KUKA KRL program: EPS_2_251806_MH56A_A_20260212042253.src

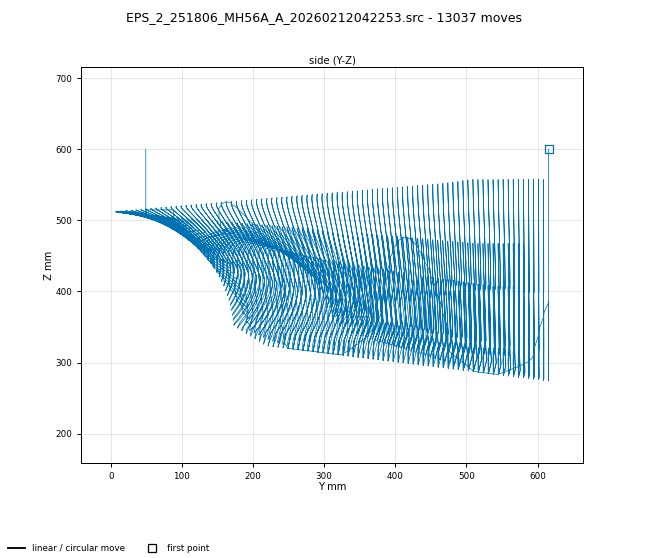
[picture p0: tool path of EPS_2_251806_MH56A_A_20260212042253.src, 13037 of 13039 moves have a stored position in this frame; points joined in program order, loops and branches not executed]
&ACCESS RVP
&REL 4
&COMMENT QRS 19112012
&PARAM EDITMASK = *
DEF PART()
EXT BAS (BAS_COMMAND :IN,REAL :IN )
INT I
BAS (#INITMOV,0 )

;KUKA QRS Post kuka4.cps  Date:22-06-2017 !

File_ID=3024

QRS_PRE_INIT()

;Init var - Until changes are made in qrs_pre_init
Outlet_Square_prg=0
Inlet_1_Square_prg=0
Inlet_2_Square_prg=0
Inlet_3_Square_prg=0
Inlet_4_Square_prg=0
Inlet_5_Square_prg=0

Outlet_1={X 0.000, Y 508.200, Z 408.000, B 0.000, E1 0.000 }
Inlet_1={X 0.000, Y 535.460, Z 257.000, B 0.000, E1 90.000 }
Inlet_2={X 0.000, Y 514.920, Z 318.000, B 0.000, E1 180.000 }
Outlet_1_type=299
Inlet_1_type=201
Inlet_2_type=299
;QRS#1=Sidecore dimensions
;QRS#2=300-12" PVC SDR 35
;QRS#3=200-8" PVC SDR 35
;QRS#4=300-12" PVC SDR 35
;QRS#5=
;QRS#6=
;QRS#7=
;QRS#8=
;QRS#9=16M PSX
;QRS#10=12-08 PSX
;QRS#11=16M PSX
;QRS#12=
;QRS#13=
;QRS#14=
;QRS#15=
;QRS#16=1220x127x838 2,75'
;QRS#17=EPS Height
;QRS#18=557,5
;QRS#19=*
;QRS#20= UPDATED VERSION 22-06-2017
;QRS#21=*
Outlet_Square=0150
Inlet_1_Square=0100
Inlet_2_Square=0150
Inlet_3_Square=0
Inlet_4_Square=0
Inlet_5_Square=0
Mill_Square=1
Outlet_Square_Prg=206
Inlet_1_Square_prg=204
Inlet_2_Square_prg=206

QRS_INIT()

$ADVANCE=5

; T1
PTP {E1 173.498,E2 173.498}
PTP {X 0,Y 615.498,A -85,B 0,C 180,E1 173.498,E2 173.498,E3 0,E4 0,E5 0,E6 0}
QRS_SPEED_INIT()
LIN {X 0,Y 615.498,Z 600,A -85,B 0,C 180,E1 173.498,E2 173.498,E3 0,E4 0,E5 0,E6 0} C_VEL
LIN {X 0,Y 615.498,Z 398.232,A -85,B 0,C 180,E1 173.498,E2 173.498} C_VEL
LIN {X 0,Y 615.498,Z 387.352,A -85,B 0,C 180,E1 173.498,E2 173.498} C_VEL
LIN {X 0,Y 615.496,Z 385.708,A -85,B 0,C 180,E1 173.418,E2 173.418} C_VEL
LIN {X 0,Y 615.498,Z 378.036,A -85,B 0,C 180,E1 172.455,E2 172.455} C_VEL
LIN {X 0,Y 615.498,Z 368.258,A -85,B 0,C 180,E1 171.463,E2 171.463} C_VEL
LIN {X 0,Y 615.498,Z 357.992,A -85,B 0,C 180,E1 170.636,E2 170.636} C_VEL
LIN {X 0,Y 615.489,Z 346.429,A -85,B 0,C 180,E1 169.889,E2 169.889} C_VEL
LIN {X 0,Y 615.479,Z 334.651,A -85,B 0,C 180,E1 169.296,E2 169.296} C_VEL
LIN {X 0,Y 615.485,Z 321.657,A -85,B 0,C 180,E1 168.807,E2 168.807} C_VEL
LIN {X 0,Y 615.492,Z 309.054,A -85,B 0,C 180,E1 168.473,E2 168.473} C_VEL
LIN {X 0,Y 615.49,Z 303.848,A -85,B 0,C 180,E1 168.369,E2 168.369} C_VEL
LIN {X 0,Y 615.48,Z 300.786,A -85,B 0,C 180,E1 166.071,E2 166.071} C_VEL
LIN {X 0,Y 615.479,Z 297.27,A -85,B 0,C 180,E1 163.413,E2 163.413} C_VEL
LIN {X 0,Y 615.488,Z 293.703,A -85,B 0,C 180,E1 160.662,E2 160.662} C_VEL
LIN {X 0,Y 615.494,Z 290.108,A -85,B 0,C 180,E1 157.864,E2 157.864} C_VEL
LIN {X 0,Y 615.499,Z 286.537,A -85,B 0,C 180,E1 155.009,E2 155.009} C_VEL
LIN {X 0,Y 615.485,Z 282.947,A -85,B 0,C 180,E1 152.085,E2 152.085} C_VEL
LIN {X 0,Y 615.497,Z 280.363,A -85,B 0,C 180,E1 149.84,E2 149.84} C_VEL
LIN {X 0,Y 615.449,Z 277.794,A -85,B 0,C 180,E1 147.54,E2 147.54} C_VEL
LIN {X 0,Y 615.456,Z 275.078,A -85,B 0,C 180,E1 145.183,E2 145.183} C_VEL
LIN {X 0,Y 615.496,Z 274.312,A -85,B 0,C 180,E1 144.166,E2 144.166} C_VEL
LIN {X 0,Y 615.481,Z 274.312,A -85,B 0,C 180,E1 141.931,E2 141.931} C_VEL
LIN {X 0,Y 615.483,Z 274.324,A -85,B 0,C 180,E1 139.393,E2 139.393} C_VEL
LIN {X 0,Y 615.467,Z 274.316,A -85,B 0,C 180,E1 136.753,E2 136.753} C_VEL
LIN {X 0,Y 615.492,Z 274.321,A -85,B 0,C 180,E1 133.998,E2 133.998} C_VEL
LIN {X 0,Y 615.443,Z 274.324,A -85,B 0,C 180,E1 131.478,E2 131.478} C_VEL
LIN {X 0,Y 615.464,Z 274.321,A -85,B 0,C 180,E1 130.609,E2 130.609} C_VEL
LIN {X 0,Y 615.478,Z 275.497,A -85,B 0,C 180,E1 129.751,E2 129.751} C_VEL
LIN {X 0,Y 615.477,Z 280.151,A -85,B 0,C 180,E1 126.935,E2 126.935} C_VEL
LIN {X 0,Y 615.455,Z 284.702,A -85,B 0,C 180,E1 124.024,E2 124.024} C_VEL
LIN {X 0,Y 615.486,Z 288.323,A -85,B 0,C 180,E1 121.686,E2 121.686} C_VEL
LIN {X 0,Y 615.494,Z 291.936,A -85,B 0,C 180,E1 119.406,E2 119.406} C_VEL
LIN {X 0,Y 615.488,Z 296.744,A -85,B 0,C 180,E1 116.444,E2 116.444} C_VEL
LIN {X 0,Y 615.478,Z 300.805,A -85,B 0,C 180,E1 114.006,E2 114.006} C_VEL
LIN {X 0,Y 615.491,Z 305.165,A -85,B 0,C 180,E1 111.432,E2 111.432} C_VEL
LIN {X 0,Y 615.488,Z 310.047,A -85,B 0,C 180,E1 108.604,E2 108.604} C_VEL
LIN {X 0,Y 615.489,Z 314.21,A -85,B 0,C 180,E1 106.3,E2 106.3} C_VEL
LIN {X 0,Y 615.499,Z 330.161,A -85,B 0,C 180,E1 106.036,E2 106.036} C_VEL
LIN {X 0,Y 615.493,Z 345.208,A -85,B 0,C 180,E1 105.65,E2 105.65} C_VEL
LIN {X 0,Y 615.479,Z 359.714,A -85,B 0,C 180,E1 105.142,E2 105.142} C_VEL
LIN {X 0,Y 615.489,Z 374.502,A -85,B 0,C 180,E1 104.473,E2 104.473} C_VEL
LIN {X 0,Y 615.496,Z 388.073,A -85,B 0,C 180,E1 103.706,E2 103.706} C_VEL
LIN {X 0,Y 615.496,Z 401.457,A -85,B 0,C 180,E1 102.782,E2 102.782} C_VEL
LIN {X 0,Y 615.495,Z 412.571,A -85,B 0,C 180,E1 101.861,E2 101.861} C_VEL
LIN {X 0,Y 615.493,Z 422.483,A -85,B 0,C 180,E1 100.89,E2 100.89} C_VEL
LIN {X 0,Y 615.495,Z 432.76,A -85,B 0,C 180,E1 99.696,E2 99.696} C_VEL
LIN {X 0,Y 615.49,Z 441.028,A -85,B 0,C 180,E1 98.537,E2 98.537} C_VEL
LIN {X 0,Y 615.491,Z 448.782,A -85,B 0,C 180,E1 97.216,E2 97.216} C_VEL
LIN {X 0,Y 615.499,Z 454.947,A -85,B 0,C 180,E1 95.899,E2 95.899} C_VEL
LIN {X 0,Y 615.489,Z 459.716,A -85,B 0,C 180,E1 94.585,E2 94.585} C_VEL
LIN {X 0,Y 615.491,Z 463.221,A -85,B 0,C 180,E1 93.273,E2 93.273} C_VEL
LIN {X 0,Y 615.5,Z 465.54,A -85,B 0,C 180,E1 91.963,E2 91.963} C_VEL
LIN {X 0,Y 615.491,Z 466.728,A -85,B 0,C 180,E1 90.654,E2 90.654} C_VEL
LIN {X 0,Y 615.492,Z 466.751,A -85,B 0,C 180,E1 89.346,E2 89.346} C_VEL
LIN {X 0,Y 615.5,Z 465.646,A -85,B 0,C 180,E1 88.037,E2 88.037} C_VEL
LIN {X 0,Y 615.494,Z 463.416,A -85,B 0,C 180,E1 86.727,E2 86.727} C_VEL
LIN {X 0,Y 615.49,Z 460.005,A -85,B 0,C 180,E1 85.416,E2 85.416} C_VEL
LIN {X 0,Y 615.499,Z 455.336,A -85,B 0,C 180,E1 84.102,E2 84.102} C_VEL
LIN {X 0,Y 615.49,Z 449.273,A -85,B 0,C 180,E1 82.785,E2 82.785} C_VEL
LIN {X 0,Y 615.493,Z 441.633,A -85,B 0,C 180,E1 81.464,E2 81.464} C_VEL
LIN {X 0,Y 615.496,Z 433.451,A -85,B 0,C 180,E1 80.304,E2 80.304} C_VEL
LIN {X 0,Y 615.495,Z 423.338,A -85,B 0,C 180,E1 79.109,E2 79.109} C_VEL
LIN {X 0,Y 615.497,Z 411.684,A -85,B 0,C 180,E1 77.972,E2 77.972} C_VEL
LIN {X 0,Y 615.498,Z 400.413,A -85,B 0,C 180,E1 77.051,E2 77.051} C_VEL
LIN {X 0,Y 615.498,Z 388.174,A -85,B 0,C 180,E1 76.21,E2 76.21} C_VEL
LIN {X 0,Y 615.495,Z 374.776,A -85,B 0,C 180,E1 75.451,E2 75.451} C_VEL
LIN {X 0,Y 615.478,Z 360.912,A -85,B 0,C 180,E1 74.816,E2 74.816} C_VEL
LIN {X 0,Y 615.496,Z 346.696,A -85,B 0,C 180,E1 74.308,E2 74.308} C_VEL
LIN {X 0,Y 615.496,Z 332.617,A -85,B 0,C 180,E1 73.931,E2 73.931} C_VEL
LIN {X 0,Y 615.494,Z 318.237,A -85,B 0,C 180,E1 73.667,E2 73.667} C_VEL
LIN {X 0,Y 615.493,Z 314.073,A -85,B 0,C 180,E1 73.601,E2 73.601} C_VEL
LIN {X 0,Y 615.489,Z 310.132,A -85,B 0,C 180,E1 71.354,E2 71.354} C_VEL
LIN {X 0,Y 615.485,Z 305.319,A -85,B 0,C 180,E1 68.568,E2 68.568} C_VEL
LIN {X 0,Y 615.48,Z 300.507,A -85,B 0,C 180,E1 65.728,E2 65.728} C_VEL
LIN {X 0,Y 615.498,Z 295.905,A -85,B 0,C 180,E1 62.953,E2 62.953} C_VEL
LIN {X 0,Y 615.477,Z 291.462,A -85,B 0,C 180,E1 60.207,E2 60.207} C_VEL
LIN {X 0,Y 615.492,Z 287.263,A -85,B 0,C 180,E1 57.543,E2 57.543} C_VEL
LIN {X 0,Y 615.477,Z 283.629,A -85,B 0,C 180,E1 55.184,E2 55.184} C_VEL
LIN {X 0,Y 615.485,Z 279.803,A -85,B 0,C 180,E1 52.758,E2 52.758} C_VEL
LIN {X 0,Y 615.484,Z 275.048,A -85,B 0,C 180,E1 49.912,E2 49.912} C_VEL
LIN {X 0,Y 615.465,Z 274.324,A -85,B 0,C 180,E1 49.392,E2 49.392} C_VEL
LIN {X 0,Y 615.463,Z 274.323,A -85,B 0,C 180,E1 46.753,E2 46.753} C_VEL
LIN {X 0,Y 615.485,Z 274.314,A -85,B 0,C 180,E1 43.997,E2 43.997} C_VEL
LIN {X 0,Y 615.467,Z 274.324,A -85,B 0,C 180,E1 41.092,E2 41.092} C_VEL
LIN {X 0,Y 615.434,Z 274.325,A -85,B 0,C 180,E1 38.908,E2 38.908} C_VEL
LIN {X 0,Y 615.483,Z 274.327,A -85,B 0,C 180,E1 36.425,E2 36.425} C_VEL
LIN {X 0,Y 615.49,Z 274.313,A -85,B 0,C 180,E1 34.022,E2 34.022} C_VEL
LIN {X 0,Y 615.47,Z 274.323,A -85,B 0,C 180,E1 31.083,E2 31.083} C_VEL
LIN {X 0,Y 615.454,Z 274.325,A -85,B 0,C 180,E1 28.445,E2 28.445} C_VEL
LIN {X 0,Y 615.461,Z 274.319,A -85,B 0,C 180,E1 25.564,E2 25.564} C_VEL
LIN {X 0,Y 615.483,Z 274.323,A -85,B 0,C 180,E1 22.845,E2 22.845} C_VEL
LIN {X 0,Y 615.496,Z 274.317,A -85,B 0,C 180,E1 20.033,E2 20.033} C_VEL
LIN {X 0,Y 615.436,Z 274.325,A -85,B 0,C 180,E1 17.272,E2 17.272} C_VEL
LIN {X 0,Y 615.493,Z 274.321,A -85,B 0,C 180,E1 14.549,E2 14.549} C_VEL
LIN {X 0,Y 615.479,Z 274.318,A -85,B 0,C 180,E1 11.861,E2 11.861} C_VEL
LIN {X 0,Y 615.458,Z 274.322,A -85,B 0,C 180,E1 9.199,E2 9.199} C_VEL
LIN {X 0,Y 615.479,Z 274.325,A -85,B 0,C 180,E1 6.557,E2 6.557} C_VEL
LIN {X 0,Y 615.461,Z 274.319,A -85,B 0,C 180,E1 3.929,E2 3.929} C_VEL
LIN {X 0,Y 615.492,Z 274.324,A -85,B 0,C 180,E1 1.309,E2 1.309} C_VEL
LIN {X 0,Y 615.484,Z 274.315,A -85,B 0,C 180,E1 -1.309,E2 -1.309} C_VEL
LIN {X 0,Y 615.458,Z 274.325,A -85,B 0,C 180,E1 -3.929,E2 -3.929} C_VEL
LIN {X 0,Y 615.462,Z 274.324,A -85,B 0,C 180,E1 -6.557,E2 -6.557} C_VEL
LIN {X 0,Y 615.492,Z 274.313,A -85,B 0,C 180,E1 -9.199,E2 -9.199} C_VEL
LIN {X 0,Y 615.489,Z 274.326,A -85,B 0,C 180,E1 -11.861,E2 -11.861} C_VEL
LIN {X 0,Y 615.437,Z 274.325,A -85,B 0,C 180,E1 -14.55,E2 -14.55} C_VEL
LIN {X 0,Y 615.491,Z 274.317,A -85,B 0,C 180,E1 -17.27,E2 -17.27} C_VEL
LIN {X 0,Y 615.484,Z 274.322,A -85,B 0,C 180,E1 -20.033,E2 -20.033} C_VEL
LIN {X 0,Y 615.477,Z 274.316,A -85,B 0,C 180,E1 -22.845,E2 -22.845} C_VEL
LIN {X 0,Y 615.446,Z 274.325,A -85,B 0,C 180,E1 -25.718,E2 -25.718} C_VEL
LIN {X 0,Y 615.448,Z 274.323,A -85,B 0,C 180,E1 -27.917,E2 -27.917} C_VEL
LIN {X 0,Y 615.492,Z 274.324,A -85,B 0,C 180,E1 -30.16,E2 -30.16} C_VEL
LIN {X 0,Y 615.473,Z 274.318,A -85,B 0,C 180,E1 -32.458,E2 -32.458} C_VEL
LIN {X 0,Y 615.487,Z 274.317,A -85,B 0,C 180,E1 -34.815,E2 -34.815} C_VEL
LIN {X 0,Y 615.457,Z 274.325,A -85,B 0,C 180,E1 -37.244,E2 -37.244} C_VEL
LIN {X 0,Y 615.485,Z 274.324,A -85,B 0,C 180,E1 -40.089,E2 -40.089} C_VEL
LIN {X 0,Y 615.488,Z 274.315,A -85,B 0,C 180,E1 -43.047,E2 -43.047} C_VEL
LIN {X 0,Y 615.449,Z 274.323,A -85,B 0,C 180,E1 -45.847,E2 -45.847} C_VEL
LIN {X 0,Y 615.496,Z 274.325,A -85,B 0,C 180,E1 -48.527,E2 -48.527} C_VEL
LIN {X 0,Y 615.468,Z 274.318,A -85,B 0,C 180,E1 -51.094,E2 -51.094} C_VEL
LIN {X 0,Y 615.483,Z 274.328,A -85,B 0,C 180,E1 -53.575,E2 -53.575} C_VEL
LIN {X 0,Y 615.468,Z 274.414,A -85,B 0,C 180,E1 -56.221,E2 -56.221} C_VEL
LIN {X 0,Y 615.492,Z 293.302,A -85,B 0,C 180,E1 -59.081,E2 -59.081} C_VEL
LIN {X 0,Y 615.485,Z 311.921,A -85,B 0,C 180,E1 -61.816,E2 -61.816} C_VEL
LIN {X 0,Y 615.492,Z 331.172,A -85,B 0,C 180,E1 -64.574,E2 -64.574} C_VEL
LIN {X 0,Y 615.499,Z 351.406,A -85,B 0,C 180,E1 -67.406,E2 -67.406} C_VEL
LIN {X 0,Y 615.485,Z 372.62,A -85,B 0,C 180,E1 -70.315,E2 -70.315} C_VEL
LIN {X 0,Y 615.491,Z 394.335,A -85,B 0,C 180,E1 -73.243,E2 -73.243} C_VEL
LIN {X 0,Y 615.484,Z 397.037,A -85,B 0,C 180,E1 -73.57,E2 -73.57} C_VEL
LIN {X 0,Y 615.478,Z 415.651,A -85,B 0,C 180,E1 -73.832,E2 -73.832} C_VEL
LIN {X 0,Y 615.491,Z 430.771,A -85,B 0,C 180,E1 -74.18,E2 -74.18} C_VEL
LIN {X 0,Y 615.493,Z 445.307,A -85,B 0,C 180,E1 -74.647,E2 -74.647} C_VEL
LIN {X 0,Y 615.497,Z 458.613,A -85,B 0,C 180,E1 -75.198,E2 -75.198} C_VEL
LIN {X 0,Y 615.498,Z 472.397,A -85,B 0,C 180,E1 -75.91,E2 -75.91} C_VEL
LIN {X 0,Y 615.498,Z 485.154,A -85,B 0,C 180,E1 -76.715,E2 -76.715} C_VEL
LIN {X 0,Y 615.496,Z 497.294,A -85,B 0,C 180,E1 -77.638,E2 -77.638} C_VEL
LIN {X 0,Y 615.497,Z 508.355,A -85,B 0,C 180,E1 -78.64,E2 -78.64} C_VEL
LIN {X 0,Y 615.496,Z 519.07,A -85,B 0,C 180,E1 -79.806,E2 -79.806} C_VEL
LIN {X 0,Y 615.495,Z 527.989,A -85,B 0,C 180,E1 -80.967,E2 -80.967} C_VEL
LIN {X 0,Y 615.492,Z 535.394,A -85,B 0,C 180,E1 -82.125,E2 -82.125} C_VEL
LIN {X 0,Y 615.491,Z 542.273,A -85,B 0,C 180,E1 -83.443,E2 -83.443} C_VEL
LIN {X 0,Y 615.491,Z 547.666,A -85,B 0,C 180,E1 -84.759,E2 -84.759} C_VEL
LIN {X 0,Y 615.491,Z 551.741,A -85,B 0,C 180,E1 -86.072,E2 -86.072} C_VEL
LIN {X 0,Y 615.496,Z 554.6,A -85,B 0,C 180,E1 -87.382,E2 -87.382} C_VEL
LIN {X 0,Y 615.493,Z 556.307,A -85,B 0,C 180,E1 -88.692,E2 -88.692} C_VEL
LIN {X 0,Y 615.491,Z 556.889,A -85,B 0,C 180,E1 -90,E2 -90} C_VEL
LIN {X 0,Y 615.493,Z 556.306,A -85,B 0,C 180,E1 -91.309,E2 -91.309} C_VEL
LIN {X 0,Y 615.496,Z 554.599,A -85,B 0,C 180,E1 -92.618,E2 -92.618} C_VEL
LIN {X 0,Y 615.491,Z 551.74,A -85,B 0,C 180,E1 -93.929,E2 -93.929} C_VEL
LIN {X 0,Y 615.491,Z 547.665,A -85,B 0,C 180,E1 -95.241,E2 -95.241} C_VEL
LIN {X 0,Y 615.491,Z 542.153,A -85,B 0,C 180,E1 -96.581,E2 -96.581} C_VEL
LIN {X 0,Y 615.492,Z 535.392,A -85,B 0,C 180,E1 -97.876,E2 -97.876} C_VEL
LIN {X 0,Y 615.495,Z 526.807,A -85,B 0,C 180,E1 -99.199,E2 -99.199} C_VEL
LIN {X 0,Y 615.494,Z 517.665,A -85,B 0,C 180,E1 -100.361,E2 -100.361} C_VEL
LIN {X 0,Y 615.497,Z 508.352,A -85,B 0,C 180,E1 -101.36,E2 -101.36} C_VEL
LIN {X 0,Y 615.496,Z 497.291,A -85,B 0,C 180,E1 -102.363,E2 -102.363} C_VEL
LIN {X 0,Y 615.498,Z 485.15,A -85,B 0,C 180,E1 -103.285,E2 -103.285} C_VEL
LIN {X 0,Y 615.498,Z 472.404,A -85,B 0,C 180,E1 -104.09,E2 -104.09} C_VEL
LIN {X 0,Y 615.497,Z 458.606,A -85,B 0,C 180,E1 -104.803,E2 -104.803} C_VEL
LIN {X 0,Y 615.495,Z 444.178,A -85,B 0,C 180,E1 -105.396,E2 -105.396} C_VEL
LIN {X 0,Y 615.488,Z 429.242,A -85,B 0,C 180,E1 -105.863,E2 -105.863} C_VEL
LIN {X 0,Y 615.478,Z 413.885,A -85,B 0,C 180,E1 -106.201,E2 -106.201} C_VEL
LIN {X 0,Y 615.485,Z 396.634,A -85,B 0,C 180,E1 -106.45,E2 -106.45} C_VEL
LIN {X 0,Y 615.484,Z 376.453,A -85,B 0,C 180,E1 -109.165,E2 -109.165} C_VEL
LIN {X 0,Y 615.481,Z 355.997,A -85,B 0,C 180,E1 -111.96,E2 -111.96} C_VEL
LIN {X 0,Y 615.498,Z 335.525,A -85,B 0,C 180,E1 -114.811,E2 -114.811} C_VEL
LIN {X 0,Y 615.497,Z 316.332,A -85,B 0,C 180,E1 -117.545,E2 -117.545} C_VEL
LIN {X 0,Y 615.489,Z 297.138,A -85,B 0,C 180,E1 -120.35,E2 -120.35} C_VEL
LIN {X 0,Y 615.485,Z 279.225,A -85,B 0,C 180,E1 -123.041,E2 -123.041} C_VEL
LIN {X 0,Y 615.477,Z 274.321,A -85,B 0,C 180,E1 -123.809,E2 -123.809} C_VEL
LIN {X 0,Y 615.458,Z 274.325,A -85,B 0,C 180,E1 -126.427,E2 -126.427} C_VEL
LIN {X 0,Y 615.486,Z 274.319,A -85,B 0,C 180,E1 -129.062,E2 -129.062} C_VEL
LIN {X 0,Y 615.465,Z 274.324,A -85,B 0,C 180,E1 -132.078,E2 -132.078} C_VEL
LIN {X 0,Y 615.476,Z 274.325,A -85,B 0,C 180,E1 -134.151,E2 -134.151} C_VEL
LIN {X 0,Y 615.492,Z 274.32,A -85,B 0,C 180,E1 -136.953,E2 -136.953} C_VEL
LIN {X 0,Y 615.458,Z 274.325,A -85,B 0,C 180,E1 -139.915,E2 -139.915} C_VEL
LIN {X 0,Y 615.483,Z 274.328,A -85,B 0,C 180,E1 -141.989,E2 -141.989} C_VEL
LIN {X 0,Y 615.469,Z 274.325,A -85,B 0,C 180,E1 -144.383,E2 -144.383} C_VEL
LIN {X 0,Y 615.49,Z 277.219,A -85,B 0,C 180,E1 -146.764,E2 -146.764} C_VEL
LIN {X 0,Y 615.489,Z 279.778,A -85,B 0,C 180,E1 -149.08,E2 -149.08} C_VEL
LIN {X 0,Y 615.494,Z 282.195,A -85,B 0,C 180,E1 -151.549,E2 -151.549} C_VEL
LIN {X 0,Y 615.478,Z 285.525,A -85,B 0,C 180,E1 -154.284,E2 -154.284} C_VEL
LIN {X 0,Y 615.473,Z 288.213,A -85,B 0,C 180,E1 -156.443,E2 -156.443} C_VEL
LIN {X 0,Y 615.479,Z 290.901,A -85,B 0,C 180,E1 -158.568,E2 -158.568} C_VEL
LIN {X 0,Y 615.483,Z 294.526,A -85,B 0,C 180,E1 -161.397,E2 -161.397} C_VEL
LIN {X 0,Y 615.477,Z 298.053,A -85,B 0,C 180,E1 -164.095,E2 -164.095} C_VEL
LIN {X 0,Y 615.494,Z 301.626,A -85,B 0,C 180,E1 -166.799,E2 -166.799} C_VEL
LIN {X 0,Y 615.488,Z 303.841,A -85,B 0,C 180,E1 -168.452,E2 -168.452} C_VEL
LIN {X 0,Y 615.49,Z 318.757,A -85,B 0,C 180,E1 -168.807,E2 -168.807} C_VEL
LIN {X 0,Y 615.478,Z 331.473,A -85,B 0,C 180,E1 -169.251,E2 -169.251} C_VEL
LIN {X 0,Y 615.488,Z 343.258,A -85,B 0,C 180,E1 -169.806,E2 -169.806} C_VEL
LIN {X 0,Y 615.498,Z 354.349,A -85,B 0,C 180,E1 -170.47,E2 -170.47} C_VEL
LIN {X 0,Y 615.498,Z 363.323,A -85,B 0,C 180,E1 -171.133,E2 -171.133} C_VEL
LIN {X 0,Y 615.498,Z 372.535,A -85,B 0,C 180,E1 -171.959,E2 -171.959} C_VEL
LIN {X 0,Y 615.499,Z 381.392,A -85,B 0,C 180,E1 -172.943,E2 -172.943} C_VEL
LIN {X 0,Y 615.497,Z 388.624,A -85,B 0,C 180,E1 -173.937,E2 -173.937} C_VEL
LIN {X 0,Y 615.497,Z 393.458,A -85,B 0,C 180,E1 -174.759,E2 -174.759} C_VEL
LIN {X 0,Y 615.497,Z 398.157,A -85,B 0,C 180,E1 -175.744,E2 -175.744} C_VEL
LIN {X 0,Y 615.495,Z 401.755,A -85,B 0,C 180,E1 -176.727,E2 -176.727} C_VEL
LIN {X 0,Y 615.496,Z 403.615,A -85,B 0,C 180,E1 -177.382,E2 -177.382} C_VEL
LIN {X 0,Y 615.497,Z 405.034,A -85,B 0,C 180,E1 -178.037,E2 -178.037} C_VEL
LIN {X 0,Y 615.497,Z 406.641,A -85,B 0,C 180,E1 -179.346,E2 -179.346} C_VEL
LIN {X 0,Y 615.494,Z 406.884,A -85,B 0,C 180,E1 -180,E2 -180} C_VEL
LIN {X 0,Y 615.495,Z 406.705,A -85,B 0,C 180,E1 -180.654,E2 -180.654} C_VEL
LIN {X 0,Y 615.496,Z 405.183,A -85,B 0,C 180,E1 -181.963,E2 -181.963} C_VEL
LIN {X 0,Y 615.498,Z 403.841,A -85,B 0,C 180,E1 -182.618,E2 -182.618} C_VEL
LIN {X 0,Y 615.497,Z 400.994,A -85,B 0,C 180,E1 -183.601,E2 -183.601} C_VEL
LIN {X 0,Y 615.498,Z 397.134,A -85,B 0,C 180,E1 -184.585,E2 -184.585} C_VEL
LIN {X 0,Y 615.498,Z 392.151,A -85,B 0,C 180,E1 -185.57,E2 -185.57} C_VEL
LIN {X 0,Y 615.496,Z 385.708,A -85,B 0,C 180,E1 -186.582,E2 -186.582} C_VEL
LIN {X 0,Y 614.829,Z 382.526,A -85,B 0,C 180,E1 -187.031,E2 -187.031} C_VEL
LIN {X 0,Y 611.989,Z 376.953,A -85,B 0,C 180,E1 -187.748,E2 -187.748} C_VEL
LIN {X 0,Y 609.138,Z 370.678,A -85,B 0,C 180,E1 -188.429,E2 -188.429} C_VEL
LIN {X 0,Y 608.477,Z 366.436,A -85,B 0,C 180,E1 -188.819,E2 -188.819} C_VEL
LIN {X 0,Y 608.493,Z 355.888,A -85,B 0,C 180,E1 -189.641,E2 -189.641} C_VEL
LIN {X 0,Y 608.49,Z 345.11,A -85,B 0,C 180,E1 -190.313,E2 -190.313} C_VEL
LIN {X 0,Y 608.505,Z 332.825,A -85,B 0,C 180,E1 -190.912,E2 -190.912} C_VEL
LIN {X 0,Y 608.525,Z 320.464,A -85,B 0,C 180,E1 -191.365,E2 -191.365} C_VEL
LIN {X 0,Y 608.55,Z 308.153,A -85,B 0,C 180,E1 -191.681,E2 -191.681} C_VEL
LIN {X 0,Y 608.436,Z 304.336,A -85,B 0,C 180,E1 -191.768,E2 -191.768} C_VEL
LIN {X 0,Y 608.43,Z 301.322,A -85,B 0,C 180,E1 -194.038,E2 -194.038} C_VEL
LIN {X 0,Y 608.414,Z 297.716,A -85,B 0,C 180,E1 -196.785,E2 -196.785} C_VEL
LIN {X 0,Y 608.415,Z 294.109,A -85,B 0,C 180,E1 -199.572,E2 -199.572} C_VEL
LIN {X 0,Y 608.432,Z 290.425,A -85,B 0,C 180,E1 -202.469,E2 -202.469} C_VEL
LIN {X 0,Y 608.43,Z 286.896,A -85,B 0,C 180,E1 -205.302,E2 -205.302} C_VEL
LIN {X 0,Y 608.434,Z 283.29,A -85,B 0,C 180,E1 -208.268,E2 -208.268} C_VEL
LIN {X 0,Y 608.418,Z 280.772,A -85,B 0,C 180,E1 -210.548,E2 -210.548} C_VEL
LIN {X 0,Y 608.446,Z 277.236,A -85,B 0,C 180,E1 -213.672,E2 -213.672} C_VEL
LIN {X 0,Y 608.409,Z 275.386,A -85,B 0,C 180,E1 -215.28,E2 -215.28} C_VEL
LIN {X 0,Y 608.471,Z 275.313,A -85,B 0,C 180,E1 -217.746,E2 -217.746} C_VEL
LIN {X 0,Y 608.449,Z 275.317,A -85,B 0,C 180,E1 -220.328,E2 -220.328} C_VEL
LIN {X 0,Y 608.437,Z 275.319,A -85,B 0,C 180,E1 -222.961,E2 -222.961} C_VEL
LIN {X 0,Y 608.461,Z 275.316,A -85,B 0,C 180,E1 -225.736,E2 -225.736} C_VEL
LIN {X 0,Y 608.474,Z 275.32,A -85,B 0,C 180,E1 -227.939,E2 -227.939} C_VEL
LIN {X 0,Y 608.424,Z 275.497,A -85,B 0,C 180,E1 -229.694,E2 -229.694} C_VEL
LIN {X 0,Y 608.448,Z 279.803,A -85,B 0,C 180,E1 -232.252,E2 -232.252} C_VEL
LIN {X 0,Y 608.398,Z 283.677,A -85,B 0,C 180,E1 -234.719,E2 -234.719} C_VEL
LIN {X 0,Y 608.437,Z 287.9,A -85,B 0,C 180,E1 -237.481,E2 -237.481} C_VEL
LIN {X 0,Y 608.427,Z 292.186,A -85,B 0,C 180,E1 -240.218,E2 -240.218} C_VEL
LIN {X 0,Y 608.435,Z 296.336,A -85,B 0,C 180,E1 -242.801,E2 -242.801} C_VEL
LIN {X 0,Y 608.424,Z 300.657,A -85,B 0,C 180,E1 -245.427,E2 -245.427} C_VEL
LIN {X 0,Y 608.435,Z 304.288,A -85,B 0,C 180,E1 -247.593,E2 -247.593} C_VEL
LIN {X 0,Y 608.426,Z 309.128,A -85,B 0,C 180,E1 -250.428,E2 -250.428} C_VEL
LIN {X 0,Y 608.418,Z 313.969,A -85,B 0,C 180,E1 -253.215,E2 -253.215} C_VEL
LIN {X 0,Y 608.427,Z 314.471,A -85,B 0,C 180,E1 -253.501,E2 -253.501} C_VEL
LIN {X 0,Y 608.679,Z 319.163,A -85,B 0,C 180,E1 -253.583,E2 -253.583} C_VEL
LIN {X 0,Y 608.672,Z 334.421,A -85,B 0,C 180,E1 -253.879,E2 -253.879} C_VEL
LIN {X 0,Y 608.624,Z 349.147,A -85,B 0,C 180,E1 -254.297,E2 -254.297} C_VEL
LIN {X 0,Y 608.603,Z 363.748,A -85,B 0,C 180,E1 -254.854,E2 -254.854} C_VEL
LIN {X 0,Y 608.574,Z 378.302,A -85,B 0,C 180,E1 -255.564,E2 -255.564} C_VEL
LIN {X 0,Y 608.554,Z 391.99,A -85,B 0,C 180,E1 -256.39,E2 -256.39} C_VEL
LIN {X 0,Y 608.528,Z 404.719,A -85,B 0,C 180,E1 -257.324,E2 -257.324} C_VEL
LIN {X 0,Y 608.497,Z 416.269,A -85,B 0,C 180,E1 -258.339,E2 -258.339} C_VEL
LIN {X 0,Y 608.475,Z 425.99,A -85,B 0,C 180,E1 -259.35,E2 -259.35} C_VEL
LIN {X 0,Y 608.477,Z 435.522,A -85,B 0,C 180,E1 -260.526,E2 -260.526} C_VEL
LIN {X 0,Y 608.457,Z 443.455,A -85,B 0,C 180,E1 -261.698,E2 -261.698} C_VEL
LIN {X 0,Y 608.44,Z 450.869,A -85,B 0,C 180,E1 -263.034,E2 -263.034} C_VEL
LIN {X 0,Y 608.45,Z 456.757,A -85,B 0,C 180,E1 -264.365,E2 -264.365} C_VEL
LIN {X 0,Y 608.425,Z 460.239,A -85,B 0,C 180,E1 -265.362,E2 -265.362} C_VEL
LIN {X 0,Y 608.42,Z 463.788,A -85,B 0,C 180,E1 -266.689,E2 -266.689} C_VEL
LIN {X 0,Y 608.444,Z 466.138,A -85,B 0,C 180,E1 -268.014,E2 -268.014} C_VEL
LIN {X 0,Y 608.434,Z 467.336,A -85,B 0,C 180,E1 -269.338,E2 -269.338} C_VEL
LIN {X 0,Y 608.435,Z 467.361,A -85,B 0,C 180,E1 -270.662,E2 -270.662} C_VEL
LIN {X 0,Y 608.444,Z 466.244,A -85,B 0,C 180,E1 -271.986,E2 -271.986} C_VEL
LIN {X 0,Y 608.423,Z 463.984,A -85,B 0,C 180,E1 -273.311,E2 -273.311} C_VEL
LIN {X 0,Y 608.425,Z 460.527,A -85,B 0,C 180,E1 -274.638,E2 -274.638} C_VEL
LIN {X 0,Y 608.437,Z 455.8,A -85,B 0,C 180,E1 -275.967,E2 -275.967} C_VEL
LIN {X 0,Y 608.456,Z 449.67,A -85,B 0,C 180,E1 -277.299,E2 -277.299} C_VEL
LIN {X 0,Y 608.468,Z 441.956,A -85,B 0,C 180,E1 -278.636,E2 -278.636} C_VEL
LIN {X 0,Y 608.472,Z 433.712,A -85,B 0,C 180,E1 -279.809,E2 -279.809} C_VEL
LIN {X 0,Y 608.476,Z 424.059,A -85,B 0,C 180,E1 -280.958,E2 -280.958} C_VEL
LIN {X 0,Y 608.509,Z 413.666,A -85,B 0,C 180,E1 -281.999,E2 -281.999} C_VEL
LIN {X 0,Y 608.533,Z 401.606,A -85,B 0,C 180,E1 -283.015,E2 -283.015} C_VEL
LIN {X 0,Y 608.564,Z 388.182,A -85,B 0,C 180,E1 -283.95,E2 -283.95} C_VEL
LIN {X 0,Y 608.602,Z 374.764,A -85,B 0,C 180,E1 -284.717,E2 -284.717} C_VEL
LIN {X 0,Y 608.595,Z 359.846,A -85,B 0,C 180,E1 -285.403,E2 -285.403} C_VEL
LIN {X 0,Y 608.644,Z 344.624,A -85,B 0,C 180,E1 -285.938,E2 -285.938} C_VEL
LIN {X 0,Y 608.671,Z 329.703,A -85,B 0,C 180,E1 -286.321,E2 -286.321} C_VEL
LIN {X 0,Y 608.582,Z 315.359,A -85,B 0,C 180,E1 -286.565,E2 -286.565} C_VEL
LIN {X 0,Y 608.453,Z 314.481,A -85,B 0,C 180,E1 -286.582,E2 -286.582} C_VEL
LIN {X 0,Y 608.434,Z 310.495,A -85,B 0,C 180,E1 -288.87,E2 -288.87} C_VEL
LIN {X 0,Y 608.414,Z 305.651,A -85,B 0,C 180,E1 -291.693,E2 -291.693} C_VEL
LIN {X 0,Y 608.422,Z 301.527,A -85,B 0,C 180,E1 -294.141,E2 -294.141} C_VEL
LIN {X 0,Y 608.432,Z 297.174,A -85,B 0,C 180,E1 -296.775,E2 -296.775} C_VEL
LIN {X 0,Y 608.445,Z 293.541,A -85,B 0,C 180,E1 -299.021,E2 -299.021} C_VEL
LIN {X 0,Y 608.447,Z 289.908,A -85,B 0,C 180,E1 -301.318,E2 -301.318} C_VEL
LIN {X 0,Y 608.449,Z 286.214,A -85,B 0,C 180,E1 -303.731,E2 -303.731} C_VEL
LIN {X 0,Y 608.446,Z 282.555,A -85,B 0,C 180,E1 -306.092,E2 -306.092} C_VEL
LIN {X 0,Y 608.431,Z 278.602,A -85,B 0,C 180,E1 -308.591,E2 -308.591} C_VEL
LIN {X 0,Y 608.433,Z 275.622,A -85,B 0,C 180,E1 -310.327,E2 -310.327} C_VEL
LIN {X 0,Y 608.465,Z 275.316,A -85,B 0,C 180,E1 -312.335,E2 -312.335} C_VEL
LIN {X 0,Y 608.449,Z 275.317,A -85,B 0,C 180,E1 -314.796,E2 -314.796} C_VEL
LIN {X 0,Y 608.451,Z 275.322,A -85,B 0,C 180,E1 -317.04,E2 -317.04} C_VEL
LIN {X 0,Y 608.423,Z 275.32,A -85,B 0,C 180,E1 -319.694,E2 -319.694} C_VEL
LIN {X 0,Y 608.457,Z 275.318,A -85,B 0,C 180,E1 -322.253,E2 -322.253} C_VEL
LIN {X 0,Y 608.439,Z 275.318,A -85,B 0,C 180,E1 -324.722,E2 -324.722} C_VEL
LIN {X 0,Y 608.451,Z 275.321,A -85,B 0,C 180,E1 -327.12,E2 -327.12} C_VEL
LIN {X 0,Y 608.472,Z 275.317,A -85,B 0,C 180,E1 -330.028,E2 -330.028} C_VEL
LIN {X 0,Y 608.419,Z 275.32,A -85,B 0,C 180,E1 -332.804,E2 -332.804} C_VEL
LIN {X 0,Y 608.452,Z 275.321,A -85,B 0,C 180,E1 -335.429,E2 -335.429} C_VEL
LIN {X 0,Y 608.477,Z 275.316,A -85,B 0,C 180,E1 -338.309,E2 -338.309} C_VEL
LIN {X 0,Y 608.438,Z 275.317,A -85,B 0,C 180,E1 -341.13,E2 -341.13} C_VEL
LIN {X 0,Y 608.446,Z 275.319,A -85,B 0,C 180,E1 -343.906,E2 -343.906} C_VEL
LIN {X 0,Y 608.459,Z 275.318,A -85,B 0,C 180,E1 -346.643,E2 -346.643} C_VEL
LIN {X 0,Y 608.459,Z 275.315,A -85,B 0,C 180,E1 -349.35,E2 -349.35} C_VEL
LIN {X 0,Y 608.468,Z 275.32,A -85,B 0,C 180,E1 -352.033,E2 -352.033} C_VEL
LIN {X 0,Y 608.428,Z 275.319,A -85,B 0,C 180,E1 -354.698,E2 -354.698} C_VEL
LIN {X 0,Y 608.483,Z 275.314,A -85,B 0,C 180,E1 -357.352,E2 -357.352} C_VEL
LIN {X 0,Y 608.479,Z 275.316,A -85,B 0,C 180,E1 -360,E2 -360} C_VEL
LIN {X 0,Y 608.441,Z 275.317,A -85,B 0,C 180,E1 -362.648,E2 -362.648} C_VEL
LIN {X 0,Y 608.469,Z 275.32,A -85,B 0,C 180,E1 -365.302,E2 -365.302} C_VEL
LIN {X 0,Y 608.436,Z 275.318,A -85,B 0,C 180,E1 -367.967,E2 -367.967} C_VEL
LIN {X 0,Y 608.457,Z 275.317,A -85,B 0,C 180,E1 -370.65,E2 -370.65} C_VEL
LIN {X 0,Y 608.462,Z 275.319,A -85,B 0,C 180,E1 -373.356,E2 -373.356} C_VEL
LIN {X 0,Y 608.419,Z 275.319,A -85,B 0,C 180,E1 -376.095,E2 -376.095} C_VEL
LIN {X 0,Y 608.46,Z 275.318,A -85,B 0,C 180,E1 -378.869,E2 -378.869} C_VEL
LIN {X 0,Y 608.466,Z 275.318,A -85,B 0,C 180,E1 -381.692,E2 -381.692} C_VEL
LIN {X 0,Y 608.436,Z 275.318,A -85,B 0,C 180,E1 -384.572,E2 -384.572} C_VEL
LIN {X 0,Y 608.434,Z 275.318,A -85,B 0,C 180,E1 -387.519,E2 -387.519} C_VEL
LIN {X 0,Y 608.459,Z 275.318,A -85,B 0,C 180,E1 -389.97,E2 -389.97} C_VEL
LIN {X 0,Y 608.456,Z 275.315,A -85,B 0,C 180,E1 -392.88,E2 -392.88} C_VEL
LIN {X 0,Y 608.426,Z 275.326,A -85,B 0,C 180,E1 -395.279,E2 -395.279} C_VEL
LIN {X 0,Y 608.413,Z 275.32,A -85,B 0,C 180,E1 -397.75,E2 -397.75} C_VEL
LIN {X 0,Y 608.452,Z 275.322,A -85,B 0,C 180,E1 -400.329,E2 -400.329} C_VEL
LIN {X 0,Y 608.453,Z 275.316,A -85,B 0,C 180,E1 -402.96,E2 -402.96} C_VEL
LIN {X 0,Y 608.426,Z 275.32,A -85,B 0,C 180,E1 -405.739,E2 -405.739} C_VEL
LIN {X 0,Y 608.421,Z 275.32,A -85,B 0,C 180,E1 -407.935,E2 -407.935} C_VEL
LIN {X 0,Y 608.444,Z 275.318,A -85,B 0,C 180,E1 -410.706,E2 -410.706} C_VEL
LIN {X 0,Y 608.449,Z 275.318,A -85,B 0,C 180,E1 -413.085,E2 -413.085} C_VEL
LIN {X 0,Y 608.448,Z 275.359,A -85,B 0,C 180,E1 -415.918,E2 -415.918} C_VEL
LIN {X 0,Y 608.788,Z 279.231,A -85,B 0,C 180,E1 -416.548,E2 -416.548} C_VEL
LIN {X 0,Y 608.725,Z 297.141,A -85,B 0,C 180,E1 -419.277,E2 -419.277} C_VEL
LIN {X 0,Y 608.669,Z 315.054,A -85,B 0,C 180,E1 -421.932,E2 -421.932} C_VEL
LIN {X 0,Y 608.638,Z 334.247,A -85,B 0,C 180,E1 -424.707,E2 -424.707} C_VEL
LIN {X 0,Y 608.588,Z 353.971,A -85,B 0,C 180,E1 -427.494,E2 -427.494} C_VEL
LIN {X 0,Y 608.541,Z 373.913,A -85,B 0,C 180,E1 -430.257,E2 -430.257} C_VEL
LIN {X 0,Y 608.526,Z 395.665,A -85,B 0,C 180,E1 -433.218,E2 -433.218} C_VEL
LIN {X 0,Y 608.52,Z 396.72,A -85,B 0,C 180,E1 -433.36,E2 -433.36} C_VEL
LIN {X 0,Y 608.669,Z 405.711,A -85,B 0,C 180,E1 -433.488,E2 -433.488} C_VEL
LIN {X 0,Y 608.666,Z 420.715,A -85,B 0,C 180,E1 -433.746,E2 -433.746} C_VEL
LIN {X 0,Y 608.644,Z 435.302,A -85,B 0,C 180,E1 -434.126,E2 -434.126} C_VEL
LIN {X 0,Y 608.613,Z 449.794,A -85,B 0,C 180,E1 -434.641,E2 -434.641} C_VEL
LIN {X 0,Y 608.602,Z 463.861,A -85,B 0,C 180,E1 -435.283,E2 -435.283} C_VEL
LIN {X 0,Y 608.562,Z 477.448,A -85,B 0,C 180,E1 -436.05,E2 -436.05} C_VEL
LIN {X 0,Y 608.547,Z 489.855,A -85,B 0,C 180,E1 -436.9,E2 -436.9} C_VEL
LIN {X 0,Y 608.522,Z 501.275,A -85,B 0,C 180,E1 -437.832,E2 -437.832} C_VEL
LIN {X 0,Y 608.491,Z 512.651,A -85,B 0,C 180,E1 -438.937,E2 -438.937} C_VEL
LIN {X 0,Y 608.471,Z 523.371,A -85,B 0,C 180,E1 -440.191,E2 -440.191} C_VEL
LIN {X 0,Y 608.468,Z 531.655,A -85,B 0,C 180,E1 -441.364,E2 -441.364} C_VEL
LIN {X 0,Y 608.457,Z 539.427,A -85,B 0,C 180,E1 -442.701,E2 -442.701} C_VEL
LIN {X 0,Y 608.437,Z 545.608,A -85,B 0,C 180,E1 -444.033,E2 -444.033} C_VEL
LIN {X 0,Y 608.427,Z 550.383,A -85,B 0,C 180,E1 -445.362,E2 -445.362} C_VEL
LIN {X 0,Y 608.421,Z 553.886,A -85,B 0,C 180,E1 -446.689,E2 -446.689} C_VEL
LIN {X 0,Y 608.444,Z 556.191,A -85,B 0,C 180,E1 -448.014,E2 -448.014} C_VEL
LIN {X 0,Y 608.436,Z 557.351,A -85,B 0,C 180,E1 -449.338,E2 -449.338} C_VEL
LIN {X 0,Y 608.436,Z 557.351,A -85,B 0,C 180,E1 -450.662,E2 -450.662} C_VEL
LIN {X 0,Y 608.444,Z 556.191,A -85,B 0,C 180,E1 -451.986,E2 -451.986} C_VEL
LIN {X 0,Y 608.421,Z 553.885,A -85,B 0,C 180,E1 -453.311,E2 -453.311} C_VEL
LIN {X 0,Y 608.427,Z 550.382,A -85,B 0,C 180,E1 -454.638,E2 -454.638} C_VEL
LIN {X 0,Y 608.437,Z 545.607,A -85,B 0,C 180,E1 -455.967,E2 -455.967} C_VEL
LIN {X 0,Y 608.457,Z 539.425,A -85,B 0,C 180,E1 -457.3,E2 -457.3} C_VEL
LIN {X 0,Y 608.468,Z 531.653,A -85,B 0,C 180,E1 -458.636,E2 -458.636} C_VEL
LIN {X 0,Y 608.471,Z 523.369,A -85,B 0,C 180,E1 -459.809,E2 -459.809} C_VEL
LIN {X 0,Y 608.493,Z 512.647,A -85,B 0,C 180,E1 -461.064,E2 -461.064} C_VEL
LIN {X 0,Y 608.522,Z 501.272,A -85,B 0,C 180,E1 -462.168,E2 -462.168} C_VEL
LIN {X 0,Y 608.547,Z 489.851,A -85,B 0,C 180,E1 -463.1,E2 -463.1} C_VEL
LIN {X 0,Y 608.563,Z 477.443,A -85,B 0,C 180,E1 -463.95,E2 -463.95} C_VEL
LIN {X 0,Y 608.602,Z 463.854,A -85,B 0,C 180,E1 -464.718,E2 -464.718} C_VEL
LIN {X 0,Y 608.613,Z 449.786,A -85,B 0,C 180,E1 -465.36,E2 -465.36} C_VEL
LIN {X 0,Y 608.67,Z 434.558,A -85,B 0,C 180,E1 -465.895,E2 -465.895} C_VEL
LIN {X 0,Y 608.662,Z 419.159,A -85,B 0,C 180,E1 -466.288,E2 -466.288} C_VEL
LIN {X 0,Y 608.69,Z 403.969,A -85,B 0,C 180,E1 -466.535,E2 -466.535} C_VEL
LIN {X 0,Y 608.531,Z 396.984,A -85,B 0,C 180,E1 -466.624,E2 -466.624} C_VEL
LIN {X 0,Y 608.546,Z 376.47,A -85,B 0,C 180,E1 -469.392,E2 -469.392} C_VEL
LIN {X 0,Y 608.569,Z 357.277,A -85,B 0,C 180,E1 -472.044,E2 -472.044} C_VEL
LIN {X 0,Y 608.645,Z 336.804,A -85,B 0,C 180,E1 -474.927,E2 -474.927} C_VEL
LIN {X 0,Y 608.675,Z 317.611,A -85,B 0,C 180,E1 -477.694,E2 -477.694} C_VEL
LIN {X 0,Y 608.716,Z 298.418,A -85,B 0,C 180,E1 -480.531,E2 -480.531} C_VEL
LIN {X 0,Y 608.759,Z 281.784,A -85,B 0,C 180,E1 -483.059,E2 -483.059} C_VEL
LIN {X 0,Y 608.886,Z 277.387,A -85,B 0,C 180,E1 -483.793,E2 -483.793} C_VEL
LIN {X 0,Y 608.443,Z 275.323,A -85,B 0,C 180,E1 -484.221,E2 -484.221} C_VEL
LIN {X 0,Y 608.48,Z 275.32,A -85,B 0,C 180,E1 -487.16,E2 -487.16} C_VEL
LIN {X 0,Y 608.478,Z 275.316,A -85,B 0,C 180,E1 -489.439,E2 -489.439} C_VEL
LIN {X 0,Y 608.449,Z 275.321,A -85,B 0,C 180,E1 -492.333,E2 -492.333} C_VEL
LIN {X 0,Y 608.441,Z 275.32,A -85,B 0,C 180,E1 -494.798,E2 -494.798} C_VEL
LIN {X 0,Y 608.458,Z 275.319,A -85,B 0,C 180,E1 -497.666,E2 -497.666} C_VEL
LIN {X 0,Y 608.446,Z 275.324,A -85,B 0,C 180,E1 -500.706,E2 -500.706} C_VEL
LIN {X 0,Y 608.457,Z 275.32,A -85,B 0,C 180,E1 -503.085,E2 -503.085} C_VEL
LIN {X 0,Y 608.435,Z 275.52,A -85,B 0,C 180,E1 -504.722,E2 -504.722} C_VEL
LIN {X 0,Y 608.457,Z 278.611,A -85,B 0,C 180,E1 -507.121,E2 -507.121} C_VEL
LIN {X 0,Y 608.457,Z 281.698,A -85,B 0,C 180,E1 -510.031,E2 -510.031} C_VEL
LIN {X 0,Y 608.427,Z 284.083,A -85,B 0,C 180,E1 -512.481,E2 -512.481} C_VEL
LIN {X 0,Y 608.43,Z 287.687,A -85,B 0,C 180,E1 -515.428,E2 -515.428} C_VEL
LIN {X 0,Y 608.412,Z 291.291,A -85,B 0,C 180,E1 -518.306,E2 -518.306} C_VEL
LIN {X 0,Y 608.415,Z 293.994,A -85,B 0,C 180,E1 -520.428,E2 -520.428} C_VEL
LIN {X 0,Y 608.416,Z 297.599,A -85,B 0,C 180,E1 -523.215,E2 -523.215} C_VEL
LIN {X 0,Y 608.422,Z 301.257,A -85,B 0,C 180,E1 -526.002,E2 -526.002} C_VEL
LIN {X 0,Y 608.426,Z 304.443,A -85,B 0,C 180,E1 -528.338,E2 -528.338} C_VEL
LIN {X 0,Y 608.541,Z 318.137,A -85,B 0,C 180,E1 -528.656,E2 -528.656} C_VEL
LIN {X 0,Y 608.514,Z 330.053,A -85,B 0,C 180,E1 -529.062,E2 -529.062} C_VEL
LIN {X 0,Y 608.498,Z 341.869,A -85,B 0,C 180,E1 -529.603,E2 -529.603} C_VEL
LIN {X 0,Y 608.501,Z 353.291,A -85,B 0,C 180,E1 -530.275,E2 -530.275} C_VEL
LIN {X 0,Y 608.474,Z 363.585,A -85,B 0,C 180,E1 -531.029,E2 -531.029} C_VEL
LIN {X 0,Y 608.464,Z 372.85,A -85,B 0,C 180,E1 -531.866,E2 -531.866} C_VEL
LIN {X 0,Y 608.466,Z 381.824,A -85,B 0,C 180,E1 -532.867,E2 -532.867} C_VEL
LIN {X 0,Y 608.444,Z 389.056,A -85,B 0,C 180,E1 -533.867,E2 -533.867} C_VEL
LIN {X 0,Y 608.462,Z 393.935,A -85,B 0,C 180,E1 -534.698,E2 -534.698} C_VEL
LIN {X 0,Y 608.441,Z 398.678,A -85,B 0,C 180,E1 -535.694,E2 -535.694} C_VEL
LIN {X 0,Y 608.425,Z 402.312,A -85,B 0,C 180,E1 -536.689,E2 -536.689} C_VEL
LIN {X 0,Y 608.425,Z 404.191,A -85,B 0,C 180,E1 -537.352,E2 -537.352} C_VEL
LIN {X 0,Y 608.442,Z 405.627,A -85,B 0,C 180,E1 -538.014,E2 -538.014} C_VEL
LIN {X 0,Y 608.44,Z 407.252,A -85,B 0,C 180,E1 -539.338,E2 -539.338} C_VEL
LIN {X 0,Y 608.434,Z 407.495,A -85,B 0,C 180,E1 -540,E2 -540} C_VEL
LIN {X 0,Y 608.438,Z 407.315,A -85,B 0,C 180,E1 -540.662,E2 -540.662} C_VEL
LIN {X 0,Y 608.441,Z 405.776,A -85,B 0,C 180,E1 -541.986,E2 -541.986} C_VEL
LIN {X 0,Y 608.426,Z 404.418,A -85,B 0,C 180,E1 -542.648,E2 -542.648} C_VEL
LIN {X 0,Y 608.45,Z 401.541,A -85,B 0,C 180,E1 -543.642,E2 -543.642} C_VEL
LIN {X 0,Y 608.433,Z 397.642,A -85,B 0,C 180,E1 -544.638,E2 -544.638} C_VEL
LIN {X 0,Y 608.45,Z 392.612,A -85,B 0,C 180,E1 -545.634,E2 -545.634} C_VEL
LIN {X 0,Y 608.441,Z 386.294,A -85,B 0,C 180,E1 -546.633,E2 -546.633} C_VEL
LIN {X 0,Y 608.476,Z 378.378,A -85,B 0,C 180,E1 -547.633,E2 -547.633} C_VEL
LIN {X 0,Y 608.472,Z 368.535,A -85,B 0,C 180,E1 -548.636,E2 -548.636} C_VEL
LIN {X 0,Y 608.477,Z 366.436,A -85,B 0,C 180,E1 -548.819,E2 -548.819} C_VEL
LIN {X 0,Y 607.81,Z 362.103,A -85,B 0,C 180,E1 -549.189,E2 -549.189} C_VEL
LIN {X 0,Y 604.969,Z 354.854,A -85,B 0,C 180,E1 -549.769,E2 -549.769} C_VEL
LIN {X 0,Y 602.144,Z 347.211,A -85,B 0,C 180,E1 -550.301,E2 -550.301} C_VEL
LIN {X 0,Y 601.508,Z 342.148,A -85,B 0,C 180,E1 -550.594,E2 -550.594} C_VEL
LIN {X 0,Y 601.51,Z 331.648,A -85,B 0,C 180,E1 -551.091,E2 -551.091} C_VEL
LIN {X 0,Y 601.57,Z 319.073,A -85,B 0,C 180,E1 -551.541,E2 -551.541} C_VEL
LIN {X 0,Y 601.514,Z 305.845,A -85,B 0,C 180,E1 -551.863,E2 -551.863} C_VEL
LIN {X 0,Y 601.336,Z 304.336,A -85,B 0,C 180,E1 -551.909,E2 -551.909} C_VEL
LIN {X 0,Y 601.323,Z 301.321,A -85,B 0,C 180,E1 -554.208,E2 -554.208} C_VEL
LIN {X 0,Y 601.335,Z 297.715,A -85,B 0,C 180,E1 -556.989,E2 -556.989} C_VEL
LIN {X 0,Y 601.316,Z 294.109,A -85,B 0,C 180,E1 -559.813,E2 -559.813} C_VEL
LIN {X 0,Y 601.336,Z 290.626,A -85,B 0,C 180,E1 -562.586,E2 -562.586} C_VEL
LIN {X 0,Y 601.35,Z 287.797,A -85,B 0,C 180,E1 -564.881,E2 -564.881} C_VEL
LIN {X 0,Y 601.35,Z 284.864,A -85,B 0,C 180,E1 -567.35,E2 -567.35} C_VEL
LIN {X 0,Y 601.339,Z 282.614,A -85,B 0,C 180,E1 -569.398,E2 -569.398} C_VEL
LIN {X 0,Y 601.312,Z 280.018,A -85,B 0,C 180,E1 -571.732,E2 -571.732} C_VEL
LIN {X 0,Y 601.358,Z 277.306,A -85,B 0,C 180,E1 -574.123,E2 -574.123} C_VEL
LIN {X 0,Y 601.337,Z 276.209,A -85,B 0,C 180,E1 -575.104,E2 -575.104} C_VEL
LIN {X 0,Y 601.438,Z 276.193,A -85,B 0,C 180,E1 -577.419,E2 -577.419} C_VEL
LIN {X 0,Y 601.415,Z 276.191,A -85,B 0,C 180,E1 -579.995,E2 -579.995} C_VEL
LIN {X 0,Y 601.409,Z 276.199,A -85,B 0,C 180,E1 -582.671,E2 -582.671} C_VEL
LIN {X 0,Y 601.401,Z 276.193,A -85,B 0,C 180,E1 -585.479,E2 -585.479} C_VEL
LIN {X 0,Y 601.405,Z 276.195,A -85,B 0,C 180,E1 -588.409,E2 -588.409} C_VEL
LIN {X 0,Y 601.372,Z 276.2,A -85,B 0,C 180,E1 -589.432,E2 -589.432} C_VEL
LIN {X 0,Y 601.414,Z 279.809,A -85,B 0,C 180,E1 -591.731,E2 -591.731} C_VEL
LIN {X 0,Y 601.367,Z 283.708,A -85,B 0,C 180,E1 -594.244,E2 -594.244} C_VEL
LIN {X 0,Y 601.351,Z 288.336,A -85,B 0,C 180,E1 -597.295,E2 -597.295} C_VEL
LIN {X 0,Y 601.359,Z 292.237,A -85,B 0,C 180,E1 -599.863,E2 -599.863} C_VEL
LIN {X 0,Y 601.35,Z 296.652,A -85,B 0,C 180,E1 -602.65,E2 -602.65} C_VEL
LIN {X 0,Y 601.351,Z 300.658,A -85,B 0,C 180,E1 -605.119,E2 -605.119} C_VEL
LIN {X 0,Y 601.338,Z 305.499,A -85,B 0,C 180,E1 -608.038,E2 -608.038} C_VEL
LIN {X 0,Y 601.328,Z 309.129,A -85,B 0,C 180,E1 -610.188,E2 -610.188} C_VEL
LIN {X 0,Y 601.34,Z 313.97,A -85,B 0,C 180,E1 -613.011,E2 -613.011} C_VEL
LIN {X 0,Y 601.36,Z 314.582,A -85,B 0,C 180,E1 -613.31,E2 -613.31} C_VEL
LIN {X 0,Y 601.889,Z 319.201,A -85,B 0,C 180,E1 -613.392,E2 -613.392} C_VEL
LIN {X 0,Y 601.861,Z 334.107,A -85,B 0,C 180,E1 -613.683,E2 -613.683} C_VEL
LIN {X 0,Y 601.769,Z 349.176,A -85,B 0,C 180,E1 -614.114,E2 -614.114} C_VEL
LIN {X 0,Y 601.742,Z 363.762,A -85,B 0,C 180,E1 -614.678,E2 -614.678} C_VEL
LIN {X 0,Y 601.658,Z 377.842,A -85,B 0,C 180,E1 -615.368,E2 -615.368} C_VEL
LIN {X 0,Y 601.616,Z 390.1,A -85,B 0,C 180,E1 -616.102,E2 -616.102} C_VEL
LIN {X 0,Y 601.545,Z 402.609,A -85,B 0,C 180,E1 -617.003,E2 -617.003} C_VEL
LIN {X 0,Y 601.487,Z 414.494,A -85,B 0,C 180,E1 -618.03,E2 -618.03} C_VEL
LIN {X 0,Y 601.433,Z 425.164,A -85,B 0,C 180,E1 -619.129,E2 -619.129} C_VEL
LIN {X 0,Y 601.41,Z 434.292,A -85,B 0,C 180,E1 -620.244,E2 -620.244} C_VEL
LIN {X 0,Y 601.402,Z 442.444,A -85,B 0,C 180,E1 -621.431,E2 -621.431} C_VEL
LIN {X 0,Y 601.366,Z 449.188,A -85,B 0,C 180,E1 -622.614,E2 -622.614} C_VEL
LIN {X 0,Y 601.357,Z 455.414,A -85,B 0,C 180,E1 -623.962,E2 -623.962} C_VEL
LIN {X 0,Y 601.328,Z 460.242,A -85,B 0,C 180,E1 -625.307,E2 -625.307} C_VEL
LIN {X 0,Y 601.336,Z 463.792,A -85,B 0,C 180,E1 -626.65,E2 -626.65} C_VEL
LIN {X 0,Y 601.343,Z 466.137,A -85,B 0,C 180,E1 -627.991,E2 -627.991} C_VEL
LIN {X 0,Y 601.334,Z 467.33,A -85,B 0,C 180,E1 -629.33,E2 -629.33} C_VEL
LIN {X 0,Y 601.335,Z 467.361,A -85,B 0,C 180,E1 -630.669,E2 -630.669} C_VEL
LIN {X 0,Y 601.343,Z 466.242,A -85,B 0,C 180,E1 -632.009,E2 -632.009} C_VEL
LIN {X 0,Y 601.339,Z 463.985,A -85,B 0,C 180,E1 -633.35,E2 -633.35} C_VEL
LIN {X 0,Y 601.328,Z 460.527,A -85,B 0,C 180,E1 -634.693,E2 -634.693} C_VEL
LIN {X 0,Y 601.358,Z 455.794,A -85,B 0,C 180,E1 -636.038,E2 -636.038} C_VEL
LIN {X 0,Y 601.365,Z 449.663,A -85,B 0,C 180,E1 -637.386,E2 -637.386} C_VEL
LIN {X 0,Y 601.389,Z 441.954,A -85,B 0,C 180,E1 -638.738,E2 -638.738} C_VEL
LIN {X 0,Y 601.428,Z 433.71,A -85,B 0,C 180,E1 -639.925,E2 -639.925} C_VEL
LIN {X 0,Y 601.443,Z 423.354,A -85,B 0,C 180,E1 -641.164,E2 -641.164} C_VEL
LIN {X 0,Y 601.503,Z 411.792,A -85,B 0,C 180,E1 -642.312,E2 -642.312} C_VEL
LIN {X 0,Y 601.56,Z 399.297,A -85,B 0,C 180,E1 -643.34,E2 -643.34} C_VEL
LIN {X 0,Y 601.641,Z 386.773,A -85,B 0,C 180,E1 -644.2,E2 -644.2} C_VEL
LIN {X 0,Y 601.715,Z 373.035,A -85,B 0,C 180,E1 -644.976,E2 -644.976} C_VEL
LIN {X 0,Y 601.749,Z 358.709,A -85,B 0,C 180,E1 -645.626,E2 -645.626} C_VEL
LIN {X 0,Y 601.816,Z 344.581,A -85,B 0,C 180,E1 -646.124,E2 -646.124} C_VEL
LIN {X 0,Y 601.871,Z 329.634,A -85,B 0,C 180,E1 -646.511,E2 -646.511} C_VEL
LIN {X 0,Y 601.792,Z 316.678,A -85,B 0,C 180,E1 -646.737,E2 -646.737} C_VEL
LIN {X 0,Y 601.336,Z 314.458,A -85,B 0,C 180,E1 -646.797,E2 -646.797} C_VEL
LIN {X 0,Y 601.333,Z 310.494,A -85,B 0,C 180,E1 -649.102,E2 -649.102} C_VEL
LIN {X 0,Y 601.341,Z 306.861,A -85,B 0,C 180,E1 -651.242,E2 -651.242} C_VEL
LIN {X 0,Y 601.347,Z 303.228,A -85,B 0,C 180,E1 -653.413,E2 -653.413} C_VEL
LIN {X 0,Y 601.359,Z 298.384,A -85,B 0,C 180,E1 -656.366,E2 -656.366} C_VEL
LIN {X 0,Y 601.363,Z 294.52,A -85,B 0,C 180,E1 -658.776,E2 -658.776} C_VEL
LIN {X 0,Y 601.37,Z 290.357,A -85,B 0,C 180,E1 -661.447,E2 -661.447} C_VEL
LIN {X 0,Y 601.372,Z 286.333,A -85,B 0,C 180,E1 -664.122,E2 -664.122} C_VEL
LIN {X 0,Y 601.393,Z 282.582,A -85,B 0,C 180,E1 -666.584,E2 -666.584} C_VEL
LIN {X 0,Y 601.409,Z 277.891,A -85,B 0,C 180,E1 -669.532,E2 -669.532} C_VEL
LIN {X 0,Y 601.345,Z 276.206,A -85,B 0,C 180,E1 -670.565,E2 -670.565} C_VEL
LIN {X 0,Y 601.406,Z 276.194,A -85,B 0,C 180,E1 -672.671,E2 -672.671} C_VEL
LIN {X 0,Y 601.399,Z 276.199,A -85,B 0,C 180,E1 -675.479,E2 -675.479} C_VEL
LIN {X 0,Y 601.422,Z 276.196,A -85,B 0,C 180,E1 -678.407,E2 -678.407} C_VEL
LIN {X 0,Y 601.398,Z 276.196,A -85,B 0,C 180,E1 -681.533,E2 -681.533} C_VEL
LIN {X 0,Y 601.406,Z 276.194,A -85,B 0,C 180,E1 -684.247,E2 -684.247} C_VEL
LIN {X 0,Y 601.426,Z 276.194,A -85,B 0,C 180,E1 -686.686,E2 -686.686} C_VEL
LIN {X 0,Y 601.4,Z 276.196,A -85,B 0,C 180,E1 -689.057,E2 -689.057} C_VEL
LIN {X 0,Y 601.375,Z 276.198,A -85,B 0,C 180,E1 -691.37,E2 -691.37} C_VEL
LIN {X 0,Y 601.4,Z 276.195,A -85,B 0,C 180,E1 -694.135,E2 -694.135} C_VEL
LIN {X 0,Y 601.395,Z 276.197,A -85,B 0,C 180,E1 -696.589,E2 -696.589} C_VEL
LIN {X 0,Y 601.422,Z 276.191,A -85,B 0,C 180,E1 -699.478,E2 -699.478} C_VEL
LIN {X 0,Y 601.373,Z 276.199,A -85,B 0,C 180,E1 -702.311,E2 -702.311} C_VEL
LIN {X 0,Y 601.39,Z 276.195,A -85,B 0,C 180,E1 -704.408,E2 -704.408} C_VEL
LIN {X 0,Y 601.421,Z 276.195,A -85,B 0,C 180,E1 -707.172,E2 -707.172} C_VEL
LIN {X 0,Y 601.438,Z 276.192,A -85,B 0,C 180,E1 -709.905,E2 -709.905} C_VEL
LIN {X 0,Y 601.373,Z 276.197,A -85,B 0,C 180,E1 -712.614,E2 -712.614} C_VEL
LIN {X 0,Y 601.424,Z 276.198,A -85,B 0,C 180,E1 -715.308,E2 -715.308} C_VEL
LIN {X 0,Y 601.417,Z 276.193,A -85,B 0,C 180,E1 -717.991,E2 -717.991} C_VEL
LIN {X 0,Y 601.439,Z 276.191,A -85,B 0,C 180,E1 -720.669,E2 -720.669} C_VEL
LIN {X 0,Y 601.418,Z 276.196,A -85,B 0,C 180,E1 -723.35,E2 -723.35} C_VEL
LIN {X 0,Y 601.383,Z 276.196,A -85,B 0,C 180,E1 -726.037,E2 -726.037} C_VEL
LIN {X 0,Y 601.439,Z 276.194,A -85,B 0,C 180,E1 -728.737,E2 -728.737} C_VEL
LIN {X 0,Y 601.435,Z 276.19,A -85,B 0,C 180,E1 -731.458,E2 -731.458} C_VEL
LIN {X 0,Y 601.377,Z 276.197,A -85,B 0,C 180,E1 -734.206,E2 -734.206} C_VEL
LIN {X 0,Y 601.409,Z 276.199,A -85,B 0,C 180,E1 -736.986,E2 -736.986} C_VEL
LIN {X 0,Y 601.406,Z 276.195,A -85,B 0,C 180,E1 -739.809,E2 -739.809} C_VEL
LIN {X 0,Y 601.412,Z 276.192,A -85,B 0,C 180,E1 -742.683,E2 -742.683} C_VEL
LIN {X 0,Y 601.389,Z 276.198,A -85,B 0,C 180,E1 -744.879,E2 -744.879} C_VEL
LIN {X 0,Y 601.392,Z 276.195,A -85,B 0,C 180,E1 -747.869,E2 -747.869} C_VEL
LIN {X 0,Y 601.428,Z 276.197,A -85,B 0,C 180,E1 -750.164,E2 -750.164} C_VEL
LIN {X 0,Y 601.416,Z 276.192,A -85,B 0,C 180,E1 -752.715,E2 -752.715} C_VEL
LIN {X 0,Y 601.39,Z 276.201,A -85,B 0,C 180,E1 -755.111,E2 -755.111} C_VEL
LIN {X 0,Y 601.392,Z 276.196,A -85,B 0,C 180,E1 -757.422,E2 -757.422} C_VEL
LIN {X 0,Y 601.397,Z 276.199,A -85,B 0,C 180,E1 -759.996,E2 -759.996} C_VEL
LIN {X 0,Y 601.411,Z 276.193,A -85,B 0,C 180,E1 -762.67,E2 -762.67} C_VEL
LIN {X 0,Y 601.398,Z 276.198,A -85,B 0,C 180,E1 -765.479,E2 -765.479} C_VEL
LIN {X 0,Y 601.415,Z 276.197,A -85,B 0,C 180,E1 -768.408,E2 -768.408} C_VEL
LIN {X 0,Y 601.431,Z 276.194,A -85,B 0,C 180,E1 -771.529,E2 -771.529} C_VEL
LIN {X 0,Y 601.388,Z 276.197,A -85,B 0,C 180,E1 -774.246,E2 -774.246} C_VEL
LIN {X 0,Y 601.449,Z 276.321,A -85,B 0,C 180,E1 -775.605,E2 -775.605} C_VEL
LIN {X 0,Y 602.124,Z 280.59,A -85,B 0,C 180,E1 -776.33,E2 -776.33} C_VEL
LIN {X 0,Y 601.958,Z 298.42,A -85,B 0,C 180,E1 -779.089,E2 -779.089} C_VEL
LIN {X 0,Y 601.854,Z 316.334,A -85,B 0,C 180,E1 -781.776,E2 -781.776} C_VEL
LIN {X 0,Y 601.792,Z 335.527,A -85,B 0,C 180,E1 -784.584,E2 -784.584} C_VEL
LIN {X 0,Y 601.687,Z 355.558,A -85,B 0,C 180,E1 -787.447,E2 -787.447} C_VEL
LIN {X 0,Y 601.615,Z 376.472,A -85,B 0,C 180,E1 -790.376,E2 -790.376} C_VEL
LIN {X 0,Y 601.551,Z 397.013,A -85,B 0,C 180,E1 -793.178,E2 -793.178} C_VEL
LIN {X 0,Y 601.88,Z 401.449,A -85,B 0,C 180,E1 -793.241,E2 -793.241} C_VEL
LIN {X 0,Y 601.838,Z 417.751,A -85,B 0,C 180,E1 -793.496,E2 -793.496} C_VEL
LIN {X 0,Y 601.809,Z 433.049,A -85,B 0,C 180,E1 -793.876,E2 -793.876} C_VEL
LIN {X 0,Y 601.766,Z 447.552,A -85,B 0,C 180,E1 -794.375,E2 -794.375} C_VEL
LIN {X 0,Y 601.693,Z 460.367,A -85,B 0,C 180,E1 -794.937,E2 -794.937} C_VEL
LIN {X 0,Y 601.641,Z 473.215,A -85,B 0,C 180,E1 -795.627,E2 -795.627} C_VEL
LIN {X 0,Y 601.565,Z 486.373,A -85,B 0,C 180,E1 -796.488,E2 -796.488} C_VEL
LIN {X 0,Y 601.531,Z 497.389,A -85,B 0,C 180,E1 -797.346,E2 -797.346} C_VEL
LIN {X 0,Y 601.494,Z 508.51,A -85,B 0,C 180,E1 -798.372,E2 -798.372} C_VEL
LIN {X 0,Y 601.441,Z 519.301,A -85,B 0,C 180,E1 -799.565,E2 -799.565} C_VEL
LIN {X 0,Y 601.406,Z 528.292,A -85,B 0,C 180,E1 -800.754,E2 -800.754} C_VEL
LIN {X 0,Y 601.403,Z 535.753,A -85,B 0,C 180,E1 -801.939,E2 -801.939} C_VEL
LIN {X 0,Y 601.366,Z 543.223,A -85,B 0,C 180,E1 -803.399,E2 -803.399} C_VEL
LIN {X 0,Y 601.353,Z 548.161,A -85,B 0,C 180,E1 -804.635,E2 -804.635} C_VEL
LIN {X 0,Y 601.338,Z 552.288,A -85,B 0,C 180,E1 -805.979,E2 -805.979} C_VEL
LIN {X 0,Y 601.323,Z 555.185,A -85,B 0,C 180,E1 -807.321,E2 -807.321} C_VEL
LIN {X 0,Y 601.345,Z 556.913,A -85,B 0,C 180,E1 -808.661,E2 -808.661} C_VEL
LIN {X 0,Y 601.332,Z 557.5,A -85,B 0,C 180,E1 -810,E2 -810} C_VEL
LIN {X 0,Y 601.345,Z 556.912,A -85,B 0,C 180,E1 -811.34,E2 -811.34} C_VEL
LIN {X 0,Y 601.323,Z 555.185,A -85,B 0,C 180,E1 -812.68,E2 -812.68} C_VEL
LIN {X 0,Y 601.338,Z 552.287,A -85,B 0,C 180,E1 -814.021,E2 -814.021} C_VEL
LIN {X 0,Y 601.353,Z 548.161,A -85,B 0,C 180,E1 -815.365,E2 -815.365} C_VEL
LIN {X 0,Y 601.354,Z 542.702,A -85,B 0,C 180,E1 -816.712,E2 -816.712} C_VEL
LIN {X 0,Y 601.403,Z 535.751,A -85,B 0,C 180,E1 -818.061,E2 -818.061} C_VEL
LIN {X 0,Y 601.393,Z 527.091,A -85,B 0,C 180,E1 -819.416,E2 -819.416} C_VEL
LIN {X 0,Y 601.439,Z 517.876,A -85,B 0,C 180,E1 -820.606,E2 -820.606} C_VEL
LIN {X 0,Y 601.494,Z 508.507,A -85,B 0,C 180,E1 -821.628,E2 -821.628} C_VEL
LIN {X 0,Y 601.531,Z 497.386,A -85,B 0,C 180,E1 -822.654,E2 -822.654} C_VEL
LIN {X 0,Y 601.595,Z 484.464,A -85,B 0,C 180,E1 -823.649,E2 -823.649} C_VEL
LIN {X 0,Y 601.664,Z 471.78,A -85,B 0,C 180,E1 -824.459,E2 -824.459} C_VEL
LIN {X 0,Y 601.72,Z 458.607,A -85,B 0,C 180,E1 -825.15,E2 -825.15} C_VEL
LIN {X 0,Y 601.768,Z 444.179,A -85,B 0,C 180,E1 -825.756,E2 -825.756} C_VEL
LIN {X 0,Y 601.83,Z 429.246,A -85,B 0,C 180,E1 -826.233,E2 -826.233} C_VEL
LIN {X 0,Y 601.855,Z 414.28,A -85,B 0,C 180,E1 -826.57,E2 -826.57} C_VEL
LIN {X 0,Y 601.745,Z 398.096,A -85,B 0,C 180,E1 -826.803,E2 -826.803} C_VEL
LIN {X 0,Y 601.548,Z 396.668,A -85,B 0,C 180,E1 -826.845,E2 -826.845} C_VEL
LIN {X 0,Y 601.594,Z 375.19,A -85,B 0,C 180,E1 -829.803,E2 -829.803} C_VEL
LIN {X 0,Y 601.705,Z 354.718,A -85,B 0,C 180,E1 -832.672,E2 -832.672} C_VEL
LIN {X 0,Y 601.782,Z 334.245,A -85,B 0,C 180,E1 -835.602,E2 -835.602} C_VEL
LIN {X 0,Y 601.854,Z 316.332,A -85,B 0,C 180,E1 -838.225,E2 -838.225} C_VEL
LIN {X 0,Y 601.959,Z 298.418,A -85,B 0,C 180,E1 -840.911,E2 -840.911} C_VEL
LIN {X 0,Y 602.088,Z 285.258,A -85,B 0,C 180,E1 -842.972,E2 -842.972} C_VEL
LIN {X 0,Y 602.281,Z 279.909,A -85,B 0,C 180,E1 -843.87,E2 -843.87} C_VEL
LIN {X 0,Y 601.432,Z 276.197,A -85,B 0,C 180,E1 -844.625,E2 -844.625} C_VEL
LIN {X 0,Y 601.436,Z 276.195,A -85,B 0,C 180,E1 -847.419,E2 -847.419} C_VEL
LIN {X 0,Y 601.413,Z 276.199,A -85,B 0,C 180,E1 -849.995,E2 -849.995} C_VEL
LIN {X 0,Y 601.411,Z 276.2,A -85,B 0,C 180,E1 -852.671,E2 -852.671} C_VEL
LIN {X 0,Y 601.399,Z 276.197,A -85,B 0,C 180,E1 -854.533,E2 -854.533} C_VEL
LIN {X 0,Y 601.415,Z 276.195,A -85,B 0,C 180,E1 -857.409,E2 -857.409} C_VEL
LIN {X 0,Y 601.402,Z 276.197,A -85,B 0,C 180,E1 -860.004,E2 -860.004} C_VEL
LIN {X 0,Y 601.436,Z 276.193,A -85,B 0,C 180,E1 -862.618,E2 -862.618} C_VEL
LIN {X 0,Y 601.382,Z 276.201,A -85,B 0,C 180,E1 -864.245,E2 -864.245} C_VEL
LIN {X 0,Y 601.406,Z 276.821,A -85,B 0,C 180,E1 -865.068,E2 -865.068} C_VEL
LIN {X 0,Y 601.425,Z 279.83,A -85,B 0,C 180,E1 -867.484,E2 -867.484} C_VEL
LIN {X 0,Y 601.409,Z 282.388,A -85,B 0,C 180,E1 -869.855,E2 -869.855} C_VEL
LIN {X 0,Y 601.369,Z 284.541,A -85,B 0,C 180,E1 -872.13,E2 -872.13} C_VEL
LIN {X 0,Y 601.339,Z 286.507,A -85,B 0,C 180,E1 -874.148,E2 -874.148} C_VEL
LIN {X 0,Y 601.336,Z 289.49,A -85,B 0,C 180,E1 -876.586,E2 -876.586} C_VEL
LIN {X 0,Y 601.345,Z 293.094,A -85,B 0,C 180,E1 -879.475,E2 -879.475} C_VEL
LIN {X 0,Y 601.309,Z 296.698,A -85,B 0,C 180,E1 -882.309,E2 -882.309} C_VEL
LIN {X 0,Y 601.318,Z 299.402,A -85,B 0,C 180,E1 -884.406,E2 -884.406} C_VEL
LIN {X 0,Y 601.319,Z 303.006,A -85,B 0,C 180,E1 -887.17,E2 -887.17} C_VEL
LIN {X 0,Y 601.336,Z 304.473,A -85,B 0,C 180,E1 -888.198,E2 -888.198} C_VEL
LIN {X 0,Y 601.606,Z 311.674,A -85,B 0,C 180,E1 -888.353,E2 -888.353} C_VEL
LIN {X 0,Y 601.568,Z 324.922,A -85,B 0,C 180,E1 -888.74,E2 -888.74} C_VEL
LIN {X 0,Y 601.516,Z 336.75,A -85,B 0,C 180,E1 -889.226,E2 -889.226} C_VEL
LIN {X 0,Y 601.498,Z 347.923,A -85,B 0,C 180,E1 -889.821,E2 -889.821} C_VEL
LIN {X 0,Y 601.456,Z 359.3,A -85,B 0,C 180,E1 -890.585,E2 -890.585} C_VEL
LIN {X 0,Y 601.424,Z 369.365,A -85,B 0,C 180,E1 -891.432,E2 -891.432} C_VEL
LIN {X 0,Y 601.418,Z 379.069,A -85,B 0,C 180,E1 -892.446,E2 -892.446} C_VEL
LIN {X 0,Y 601.377,Z 386.389,A -85,B 0,C 180,E1 -893.393,E2 -893.393} C_VEL
LIN {X 0,Y 601.372,Z 392.112,A -85,B 0,C 180,E1 -894.299,E2 -894.299} C_VEL
LIN {X 0,Y 601.335,Z 397.254,A -85,B 0,C 180,E1 -895.307,E2 -895.307} C_VEL
LIN {X 0,Y 601.368,Z 401.244,A -85,B 0,C 180,E1 -896.315,E2 -896.315} C_VEL
LIN {X 0,Y 601.324,Z 404.193,A -85,B 0,C 180,E1 -897.321,E2 -897.321} C_VEL
LIN {X 0,Y 601.341,Z 405.627,A -85,B 0,C 180,E1 -897.991,E2 -897.991} C_VEL
LIN {X 0,Y 601.34,Z 407.253,A -85,B 0,C 180,E1 -899.33,E2 -899.33} C_VEL
LIN {X 0,Y 601.335,Z 407.496,A -85,B 0,C 180,E1 -900,E2 -900} C_VEL
LIN {X 0,Y 601.339,Z 407.315,A -85,B 0,C 180,E1 -900.67,E2 -900.67} C_VEL
LIN {X 0,Y 601.34,Z 405.776,A -85,B 0,C 180,E1 -902.009,E2 -902.009} C_VEL
LIN {X 0,Y 601.326,Z 404.417,A -85,B 0,C 180,E1 -902.68,E2 -902.68} C_VEL
LIN {X 0,Y 601.368,Z 401.54,A -85,B 0,C 180,E1 -903.685,E2 -903.685} C_VEL
LIN {X 0,Y 601.337,Z 397.64,A -85,B 0,C 180,E1 -904.693,E2 -904.693} C_VEL
LIN {X 0,Y 601.373,Z 392.61,A -85,B 0,C 180,E1 -905.701,E2 -905.701} C_VEL
LIN {X 0,Y 601.382,Z 386.291,A -85,B 0,C 180,E1 -906.711,E2 -906.711} C_VEL
LIN {X 0,Y 601.396,Z 378.374,A -85,B 0,C 180,E1 -907.723,E2 -907.723} C_VEL
LIN {X 0,Y 601.437,Z 368.529,A -85,B 0,C 180,E1 -908.738,E2 -908.738} C_VEL
LIN {X 0,Y 601.448,Z 358.206,A -85,B 0,C 180,E1 -909.585,E2 -909.585} C_VEL
LIN {X 0,Y 601.491,Z 346.587,A -85,B 0,C 180,E1 -910.349,E2 -910.349} C_VEL
LIN {X 0,Y 601.508,Z 342.148,A -85,B 0,C 180,E1 -910.594,E2 -910.594} C_VEL
LIN {X 0,Y 600.882,Z 337.02,A -85,B 0,C 180,E1 -910.869,E2 -910.869} C_VEL
LIN {X 0,Y 598.107,Z 328.565,A -85,B 0,C 180,E1 -911.288,E2 -911.288} C_VEL
LIN {X 0,Y 595.316,Z 319.814,A -85,B 0,C 180,E1 -911.643,E2 -911.643} C_VEL
LIN {X 0,Y 594.661,Z 314.226,A -85,B 0,C 180,E1 -911.814,E2 -911.814} C_VEL
LIN {X 0,Y 594.444,Z 305.816,A -85,B 0,C 180,E1 -912.006,E2 -912.006} C_VEL
LIN {X 0,Y 594.258,Z 304.335,A -85,B 0,C 180,E1 -912.053,E2 -912.053} C_VEL
LIN {X 0,Y 594.239,Z 301.32,A -85,B 0,C 180,E1 -914.381,E2 -914.381} C_VEL
LIN {X 0,Y 594.236,Z 297.714,A -85,B 0,C 180,E1 -917.198,E2 -917.198} C_VEL
LIN {X 0,Y 594.223,Z 294.108,A -85,B 0,C 180,E1 -920.059,E2 -920.059} C_VEL
LIN {X 0,Y 594.247,Z 290.826,A -85,B 0,C 180,E1 -922.707,E2 -922.707} C_VEL
LIN {X 0,Y 594.256,Z 287.796,A -85,B 0,C 180,E1 -925.199,E2 -925.199} C_VEL
LIN {X 0,Y 594.303,Z 284.561,A -85,B 0,C 180,E1 -928.231,E2 -928.231} C_VEL
LIN {X 0,Y 594.258,Z 281.909,A -85,B 0,C 180,E1 -930.567,E2 -930.567} C_VEL
LIN {X 0,Y 594.251,Z 279.227,A -85,B 0,C 180,E1 -932.958,E2 -932.958} C_VEL
LIN {X 0,Y 594.279,Z 277.385,A -85,B 0,C 180,E1 -934.587,E2 -934.587} C_VEL
LIN {X 0,Y 594.369,Z 277.069,A -85,B 0,C 180,E1 -936.481,E2 -936.481} C_VEL
LIN {X 0,Y 594.391,Z 277.072,A -85,B 0,C 180,E1 -938.805,E2 -938.805} C_VEL
LIN {X 0,Y 594.383,Z 277.067,A -85,B 0,C 180,E1 -941.848,E2 -941.848} C_VEL
LIN {X 0,Y 594.362,Z 277.076,A -85,B 0,C 180,E1 -944.238,E2 -944.238} C_VEL
LIN {X 0,Y 594.339,Z 277.073,A -85,B 0,C 180,E1 -947.151,E2 -947.151} C_VEL
LIN {X 0,Y 594.345,Z 277.076,A -85,B 0,C 180,E1 -949.431,E2 -949.431} C_VEL
LIN {X 0,Y 594.375,Z 279.993,A -85,B 0,C 180,E1 -951.297,E2 -951.297} C_VEL
LIN {X 0,Y 594.335,Z 283.774,A -85,B 0,C 180,E1 -953.754,E2 -953.754} C_VEL
LIN {X 0,Y 594.27,Z 287.485,A -85,B 0,C 180,E1 -956.231,E2 -956.231} C_VEL
LIN {X 0,Y 594.319,Z 291.09,A -85,B 0,C 180,E1 -958.647,E2 -958.647} C_VEL
LIN {X 0,Y 594.299,Z 295.819,A -85,B 0,C 180,E1 -961.769,E2 -961.769} C_VEL
LIN {X 0,Y 594.296,Z 299.449,A -85,B 0,C 180,E1 -964.052,E2 -964.052} C_VEL
LIN {X 0,Y 594.29,Z 304.29,A -85,B 0,C 180,E1 -967.029,E2 -967.029} C_VEL
LIN {X 0,Y 594.236,Z 309.13,A -85,B 0,C 180,E1 -969.941,E2 -969.941} C_VEL
LIN {X 0,Y 594.233,Z 312.761,A -85,B 0,C 180,E1 -972.091,E2 -972.091} C_VEL
LIN {X 0,Y 594.268,Z 314.473,A -85,B 0,C 180,E1 -973.096,E2 -973.096} C_VEL
LIN {X 0,Y 595.093,Z 319.239,A -85,B 0,C 180,E1 -973.197,E2 -973.197} C_VEL
LIN {X 0,Y 595.046,Z 334.133,A -85,B 0,C 180,E1 -973.491,E2 -973.491} C_VEL
LIN {X 0,Y 594.933,Z 349.204,A -85,B 0,C 180,E1 -973.926,E2 -973.926} C_VEL
LIN {X 0,Y 594.865,Z 363.775,A -85,B 0,C 180,E1 -974.496,E2 -974.496} C_VEL
LIN {X 0,Y 594.738,Z 377.851,A -85,B 0,C 180,E1 -975.194,E2 -975.194} C_VEL
LIN {X 0,Y 594.676,Z 390.639,A -85,B 0,C 180,E1 -975.972,E2 -975.972} C_VEL
LIN {X 0,Y 594.554,Z 403.677,A -85,B 0,C 180,E1 -976.934,E2 -976.934} C_VEL
LIN {X 0,Y 594.49,Z 414.494,A -85,B 0,C 180,E1 -977.887,E2 -977.887} C_VEL
LIN {X 0,Y 594.403,Z 424.498,A -85,B 0,C 180,E1 -978.921,E2 -978.921} C_VEL
LIN {X 0,Y 594.369,Z 434.299,A -85,B 0,C 180,E1 -980.128,E2 -980.128} C_VEL
LIN {X 0,Y 594.341,Z 442.445,A -85,B 0,C 180,E1 -981.328,E2 -981.328} C_VEL
LIN {X 0,Y 594.287,Z 449.194,A -85,B 0,C 180,E1 -982.525,E2 -982.525} C_VEL
LIN {X 0,Y 594.279,Z 455.414,A -85,B 0,C 180,E1 -983.89,E2 -983.89} C_VEL
LIN {X 0,Y 594.23,Z 460.246,A -85,B 0,C 180,E1 -985.251,E2 -985.251} C_VEL
LIN {X 0,Y 594.256,Z 463.796,A -85,B 0,C 180,E1 -986.61,E2 -986.61} C_VEL
LIN {X 0,Y 594.241,Z 466.136,A -85,B 0,C 180,E1 -987.967,E2 -987.967} C_VEL
LIN {X 0,Y 594.235,Z 467.324,A -85,B 0,C 180,E1 -989.322,E2 -989.322} C_VEL
LIN {X 0,Y 594.236,Z 467.356,A -85,B 0,C 180,E1 -990.677,E2 -990.677} C_VEL
LIN {X 0,Y 594.242,Z 466.24,A -85,B 0,C 180,E1 -992.033,E2 -992.033} C_VEL
LIN {X 0,Y 594.258,Z 463.987,A -85,B 0,C 180,E1 -993.39,E2 -993.39} C_VEL
LIN {X 0,Y 594.231,Z 460.527,A -85,B 0,C 180,E1 -994.749,E2 -994.749} C_VEL
LIN {X 0,Y 594.279,Z 455.787,A -85,B 0,C 180,E1 -996.11,E2 -996.11} C_VEL
LIN {X 0,Y 594.287,Z 449.653,A -85,B 0,C 180,E1 -997.474,E2 -997.474} C_VEL
LIN {X 0,Y 594.332,Z 441.951,A -85,B 0,C 180,E1 -998.843,E2 -998.843} C_VEL
LIN {X 0,Y 594.387,Z 433.706,A -85,B 0,C 180,E1 -1000.044,E2 -1000.044} C_VEL
LIN {X 0,Y 594.41,Z 423.963,A -85,B 0,C 180,E1 -1001.229,E2 -1001.229} C_VEL
LIN {X 0,Y 594.516,Z 413.64,A -85,B 0,C 180,E1 -1002.285,E2 -1002.285} C_VEL
LIN {X 0,Y 594.579,Z 401.593,A -85,B 0,C 180,E1 -1003.326,E2 -1003.326} C_VEL
LIN {X 0,Y 594.683,Z 388.103,A -85,B 0,C 180,E1 -1004.285,E2 -1004.285} C_VEL
LIN {X 0,Y 594.789,Z 374.718,A -85,B 0,C 180,E1 -1005.067,E2 -1005.067} C_VEL
LIN {X 0,Y 594.876,Z 359.815,A -85,B 0,C 180,E1 -1005.767,E2 -1005.767} C_VEL
LIN {X 0,Y 594.984,Z 345.262,A -85,B 0,C 180,E1 -1006.292,E2 -1006.292} C_VEL
LIN {X 0,Y 595.06,Z 330.274,A -85,B 0,C 180,E1 -1006.69,E2 -1006.69} C_VEL
LIN {X 0,Y 595.003,Z 318.096,A -85,B 0,C 180,E1 -1006.913,E2 -1006.913} C_VEL
LIN {X 0,Y 594.258,Z 314.483,A -85,B 0,C 180,E1 -1006.988,E2 -1006.988} C_VEL
LIN {X 0,Y 594.254,Z 310.493,A -85,B 0,C 180,E1 -1009.338,E2 -1009.338} C_VEL
LIN {X 0,Y 594.268,Z 306.86,A -85,B 0,C 180,E1 -1011.507,E2 -1011.507} C_VEL
LIN {X 0,Y 594.253,Z 303.227,A -85,B 0,C 180,E1 -1013.71,E2 -1013.71} C_VEL
LIN {X 0,Y 594.288,Z 298.383,A -85,B 0,C 180,E1 -1016.704,E2 -1016.704} C_VEL
LIN {X 0,Y 594.293,Z 294.75,A -85,B 0,C 180,E1 -1019.003,E2 -1019.003} C_VEL
LIN {X 0,Y 594.305,Z 290.814,A -85,B 0,C 180,E1 -1021.631,E2 -1021.631} C_VEL
LIN {X 0,Y 594.315,Z 286.403,A -85,B 0,C 180,E1 -1024.584,E2 -1024.584} C_VEL
LIN {X 0,Y 594.332,Z 282.639,A -85,B 0,C 180,E1 -1027.09,E2 -1027.09} C_VEL
LIN {X 0,Y 594.369,Z 278.483,A -85,B 0,C 180,E1 -1029.681,E2 -1029.681} C_VEL
LIN {X 0,Y 594.322,Z 277.081,A -85,B 0,C 180,E1 -1030.571,E2 -1030.571} C_VEL
LIN {X 0,Y 594.358,Z 277.072,A -85,B 0,C 180,E1 -1032.851,E2 -1032.851} C_VEL
LIN {X 0,Y 594.346,Z 277.079,A -85,B 0,C 180,E1 -1035.193,E2 -1035.193} C_VEL
LIN {X 0,Y 594.363,Z 277.071,A -85,B 0,C 180,E1 -1037.624,E2 -1037.624} C_VEL
LIN {X 0,Y 594.359,Z 277.078,A -85,B 0,C 180,E1 -1040.318,E2 -1040.318} C_VEL
LIN {X 0,Y 594.359,Z 277.071,A -85,B 0,C 180,E1 -1042.911,E2 -1042.911} C_VEL
LIN {X 0,Y 594.385,Z 277.069,A -85,B 0,C 180,E1 -1045.861,E2 -1045.861} C_VEL
LIN {X 0,Y 594.367,Z 277.077,A -85,B 0,C 180,E1 -1048.649,E2 -1048.649} C_VEL
LIN {X 0,Y 594.337,Z 277.074,A -85,B 0,C 180,E1 -1051.05,E2 -1051.05} C_VEL
LIN {X 0,Y 594.361,Z 277.072,A -85,B 0,C 180,E1 -1054.055,E2 -1054.055} C_VEL
LIN {X 0,Y 594.378,Z 277.069,A -85,B 0,C 180,E1 -1056.295,E2 -1056.295} C_VEL
LIN {X 0,Y 594.394,Z 277.067,A -85,B 0,C 180,E1 -1059.224,E2 -1059.224} C_VEL
LIN {X 0,Y 594.328,Z 277.079,A -85,B 0,C 180,E1 -1062.094,E2 -1062.094} C_VEL
LIN {X 0,Y 594.345,Z 277.073,A -85,B 0,C 180,E1 -1064.218,E2 -1064.218} C_VEL
LIN {X 0,Y 594.378,Z 277.069,A -85,B 0,C 180,E1 -1066.321,E2 -1066.321} C_VEL
LIN {X 0,Y 594.373,Z 277.07,A -85,B 0,C 180,E1 -1069.095,E2 -1069.095} C_VEL
LIN {X 0,Y 594.378,Z 277.075,A -85,B 0,C 180,E1 -1071.843,E2 -1071.843} C_VEL
LIN {X 0,Y 594.36,Z 277.07,A -85,B 0,C 180,E1 -1074.572,E2 -1074.572} C_VEL
LIN {X 0,Y 594.413,Z 277.067,A -85,B 0,C 180,E1 -1077.289,E2 -1077.289} C_VEL
LIN {X 0,Y 594.416,Z 277.067,A -85,B 0,C 180,E1 -1080,E2 -1080} C_VEL
LIN {X 0,Y 594.38,Z 277.069,A -85,B 0,C 180,E1 -1082.711,E2 -1082.711} C_VEL
LIN {X 0,Y 594.39,Z 277.071,A -85,B 0,C 180,E1 -1085.428,E2 -1085.428} C_VEL
LIN {X 0,Y 594.366,Z 277.072,A -85,B 0,C 180,E1 -1088.157,E2 -1088.157} C_VEL
LIN {X 0,Y 594.387,Z 277.066,A -85,B 0,C 180,E1 -1091.072,E2 -1091.072} C_VEL
LIN {X 0,Y 594.362,Z 277.077,A -85,B 0,C 180,E1 -1093.679,E2 -1093.679} C_VEL
LIN {X 0,Y 594.359,Z 277.075,A -85,B 0,C 180,E1 -1096.708,E2 -1096.708} C_VEL
LIN {X 0,Y 594.37,Z 277.07,A -85,B 0,C 180,E1 -1099.334,E2 -1099.334} C_VEL
LIN {X 0,Y 594.361,Z 277.072,A -85,B 0,C 180,E1 -1101.503,E2 -1101.503} C_VEL
LIN {X 0,Y 594.366,Z 277.076,A -85,B 0,C 180,E1 -1103.705,E2 -1103.705} C_VEL
LIN {X 0,Y 594.368,Z 277.074,A -85,B 0,C 180,E1 -1106.7,E2 -1106.7} C_VEL
LIN {X 0,Y 594.381,Z 277.07,A -85,B 0,C 180,E1 -1108.998,E2 -1108.998} C_VEL
LIN {X 0,Y 594.383,Z 277.072,A -85,B 0,C 180,E1 -1111.643,E2 -1111.643} C_VEL
LIN {X 0,Y 594.378,Z 277.069,A -85,B 0,C 180,E1 -1114.58,E2 -1114.58} C_VEL
LIN {X 0,Y 594.356,Z 277.072,A -85,B 0,C 180,E1 -1117.604,E2 -1117.604} C_VEL
LIN {X 0,Y 594.37,Z 277.072,A -85,B 0,C 180,E1 -1120.567,E2 -1120.567} C_VEL
LIN {X 0,Y 594.366,Z 277.074,A -85,B 0,C 180,E1 -1123.299,E2 -1123.299} C_VEL
LIN {X 0,Y 594.359,Z 277.071,A -85,B 0,C 180,E1 -1126.161,E2 -1126.161} C_VEL
LIN {X 0,Y 594.368,Z 277.071,A -85,B 0,C 180,E1 -1129.179,E2 -1129.179} C_VEL
LIN {X 0,Y 594.388,Z 277.075,A -85,B 0,C 180,E1 -1132.059,E2 -1132.059} C_VEL
LIN {X 0,Y 594.416,Z 277.069,A -85,B 0,C 180,E1 -1135.217,E2 -1135.217} C_VEL
LIN {X 0,Y 595.426,Z 282.033,A -85,B 0,C 180,E1 -1136.117,E2 -1136.117} C_VEL
LIN {X 0,Y 595.236,Z 298.42,A -85,B 0,C 180,E1 -1138.701,E2 -1138.701} C_VEL
LIN {X 0,Y 595.086,Z 316.334,A -85,B 0,C 180,E1 -1141.425,E2 -1141.425} C_VEL
LIN {X 0,Y 594.938,Z 336.806,A -85,B 0,C 180,E1 -1144.458,E2 -1144.458} C_VEL
LIN {X 0,Y 594.779,Z 356.355,A -85,B 0,C 180,E1 -1147.284,E2 -1147.284} C_VEL
LIN {X 0,Y 594.673,Z 377.752,A -85,B 0,C 180,E1 -1150.317,E2 -1150.317} C_VEL
LIN {X 0,Y 594.536,Z 396.797,A -85,B 0,C 180,E1 -1152.968,E2 -1152.968} C_VEL
LIN {X 0,Y 595.095,Z 401.618,A -85,B 0,C 180,E1 -1153.047,E2 -1153.047} C_VEL
LIN {X 0,Y 595.034,Z 417.884,A -85,B 0,C 180,E1 -1153.304,E2 -1153.304} C_VEL
LIN {X 0,Y 594.991,Z 433.049,A -85,B 0,C 180,E1 -1153.686,E2 -1153.686} C_VEL
LIN {X 0,Y 594.925,Z 447.554,A -85,B 0,C 180,E1 -1154.19,E2 -1154.19} C_VEL
LIN {X 0,Y 594.816,Z 460.37,A -85,B 0,C 180,E1 -1154.758,E2 -1154.758} C_VEL
LIN {X 0,Y 594.696,Z 474.628,A -85,B 0,C 180,E1 -1155.543,E2 -1155.543} C_VEL
LIN {X 0,Y 594.606,Z 487.535,A -85,B 0,C 180,E1 -1156.414,E2 -1156.414} C_VEL
LIN {X 0,Y 594.519,Z 499.337,A -85,B 0,C 180,E1 -1157.368,E2 -1157.368} C_VEL
LIN {X 0,Y 594.442,Z 510.141,A -85,B 0,C 180,E1 -1158.405,E2 -1158.405} C_VEL
LIN {X 0,Y 594.396,Z 520.662,A -85,B 0,C 180,E1 -1159.612,E2 -1159.612} C_VEL
LIN {X 0,Y 594.34,Z 529.414,A -85,B 0,C 180,E1 -1160.814,E2 -1160.814} C_VEL
LIN {X 0,Y 594.323,Z 535.753,A -85,B 0,C 180,E1 -1161.842,E2 -1161.842} C_VEL
LIN {X 0,Y 594.275,Z 542.704,A -85,B 0,C 180,E1 -1163.208,E2 -1163.208} C_VEL
LIN {X 0,Y 594.274,Z 548.161,A -85,B 0,C 180,E1 -1164.571,E2 -1164.571} C_VEL
LIN {X 0,Y 594.251,Z 552.289,A -85,B 0,C 180,E1 -1165.931,E2 -1165.931} C_VEL
LIN {X 0,Y 594.223,Z 555.186,A -85,B 0,C 180,E1 -1167.289,E2 -1167.289} C_VEL
LIN {X 0,Y 594.245,Z 556.913,A -85,B 0,C 180,E1 -1168.645,E2 -1168.645} C_VEL
LIN {X 0,Y 594.233,Z 557.5,A -85,B 0,C 180,E1 -1170,E2 -1170} C_VEL
LIN {X 0,Y 594.245,Z 556.912,A -85,B 0,C 180,E1 -1171.356,E2 -1171.356} C_VEL
LIN {X 0,Y 594.223,Z 555.185,A -85,B 0,C 180,E1 -1172.712,E2 -1172.712} C_VEL
LIN {X 0,Y 594.251,Z 552.288,A -85,B 0,C 180,E1 -1174.069,E2 -1174.069} C_VEL
LIN {X 0,Y 594.274,Z 548.161,A -85,B 0,C 180,E1 -1175.429,E2 -1175.429} C_VEL
LIN {X 0,Y 594.275,Z 542.702,A -85,B 0,C 180,E1 -1176.792,E2 -1176.792} C_VEL
LIN {X 0,Y 594.323,Z 535.75,A -85,B 0,C 180,E1 -1178.158,E2 -1178.158} C_VEL
LIN {X 0,Y 594.341,Z 527.09,A -85,B 0,C 180,E1 -1179.529,E2 -1179.529} C_VEL
LIN {X 0,Y 594.402,Z 517.875,A -85,B 0,C 180,E1 -1180.733,E2 -1180.733} C_VEL
LIN {X 0,Y 594.467,Z 508.507,A -85,B 0,C 180,E1 -1181.767,E2 -1181.767} C_VEL
LIN {X 0,Y 594.552,Z 497.386,A -85,B 0,C 180,E1 -1182.805,E2 -1182.805} C_VEL
LIN {X 0,Y 594.652,Z 484.644,A -85,B 0,C 180,E1 -1183.799,E2 -1183.799} C_VEL
LIN {X 0,Y 594.748,Z 471.779,A -85,B 0,C 180,E1 -1184.631,E2 -1184.631} C_VEL
LIN {X 0,Y 594.832,Z 458.604,A -85,B 0,C 180,E1 -1185.329,E2 -1185.329} C_VEL
LIN {X 0,Y 594.922,Z 444.178,A -85,B 0,C 180,E1 -1185.942,E2 -1185.942} C_VEL
LIN {X 0,Y 595.002,Z 429.246,A -85,B 0,C 180,E1 -1186.424,E2 -1186.424} C_VEL
LIN {X 0,Y 595.041,Z 413.983,A -85,B 0,C 180,E1 -1186.771,E2 -1186.771} C_VEL
LIN {X 0,Y 594.933,Z 398.813,A -85,B 0,C 180,E1 -1186.993,E2 -1186.993} C_VEL
LIN {X 0,Y 594.524,Z 396.643,A -85,B 0,C 180,E1 -1187.054,E2 -1187.054} C_VEL
LIN {X 0,Y 594.665,Z 376.47,A -85,B 0,C 180,E1 -1189.864,E2 -1189.864} C_VEL
LIN {X 0,Y 594.798,Z 355.519,A -85,B 0,C 180,E1 -1192.835,E2 -1192.835} C_VEL
LIN {X 0,Y 594.932,Z 335.525,A -85,B 0,C 180,E1 -1195.73,E2 -1195.73} C_VEL
LIN {X 0,Y 595.055,Z 317.611,A -85,B 0,C 180,E1 -1198.384,E2 -1198.384} C_VEL
LIN {X 0,Y 595.204,Z 299.698,A -85,B 0,C 180,E1 -1201.104,E2 -1201.104} C_VEL
LIN {X 0,Y 595.506,Z 286.133,A -85,B 0,C 180,E1 -1203.304,E2 -1203.304} C_VEL
LIN {X 0,Y 595.552,Z 281.611,A -85,B 0,C 180,E1 -1204.096,E2 -1204.096} C_VEL
LIN {X 0,Y 594.374,Z 277.075,A -85,B 0,C 180,E1 -1205.075,E2 -1205.075} C_VEL
LIN {X 0,Y 594.379,Z 277.072,A -85,B 0,C 180,E1 -1207.942,E2 -1207.942} C_VEL
LIN {X 0,Y 594.371,Z 277.074,A -85,B 0,C 180,E1 -1210.821,E2 -1210.821} C_VEL
LIN {X 0,Y 594.377,Z 277.076,A -85,B 0,C 180,E1 -1213.84,E2 -1213.84} C_VEL
LIN {X 0,Y 594.369,Z 277.077,A -85,B 0,C 180,E1 -1216.701,E2 -1216.701} C_VEL
LIN {X 0,Y 594.358,Z 277.078,A -85,B 0,C 180,E1 -1219.432,E2 -1219.432} C_VEL
LIN {X 0,Y 594.391,Z 277.072,A -85,B 0,C 180,E1 -1222.392,E2 -1222.392} C_VEL
LIN {X 0,Y 594.317,Z 277.18,A -85,B 0,C 180,E1 -1224.682,E2 -1224.682} C_VEL
LIN {X 0,Y 594.371,Z 280.234,A -85,B 0,C 180,E1 -1227.09,E2 -1227.09} C_VEL
LIN {X 0,Y 594.374,Z 283.006,A -85,B 0,C 180,E1 -1229.674,E2 -1229.674} C_VEL
LIN {X 0,Y 594.363,Z 285.116,A -85,B 0,C 180,E1 -1231.772,E2 -1231.772} C_VEL
LIN {X 0,Y 594.278,Z 286.999,A -85,B 0,C 180,E1 -1234.051,E2 -1234.051} C_VEL
LIN {X 0,Y 594.241,Z 289.49,A -85,B 0,C 180,E1 -1236.29,E2 -1236.29} C_VEL
LIN {X 0,Y 594.293,Z 293.095,A -85,B 0,C 180,E1 -1239.22,E2 -1239.22} C_VEL
LIN {X 0,Y 594.207,Z 296.699,A -85,B 0,C 180,E1 -1242.09,E2 -1242.09} C_VEL
LIN {X 0,Y 594.245,Z 299.402,A -85,B 0,C 180,E1 -1244.216,E2 -1244.216} C_VEL
LIN {X 0,Y 594.237,Z 303.007,A -85,B 0,C 180,E1 -1247.014,E2 -1247.014} C_VEL
LIN {X 0,Y 594.251,Z 304.502,A -85,B 0,C 180,E1 -1248.055,E2 -1248.055} C_VEL
LIN {X 0,Y 594.647,Z 308.953,A -85,B 0,C 180,E1 -1248.15,E2 -1248.15} C_VEL
LIN {X 0,Y 594.601,Z 321.61,A -85,B 0,C 180,E1 -1248.494,E2 -1248.494} C_VEL
LIN {X 0,Y 594.531,Z 334.034,A -85,B 0,C 180,E1 -1248.972,E2 -1248.972} C_VEL
LIN {X 0,Y 594.514,Z 345.026,A -85,B 0,C 180,E1 -1249.528,E2 -1249.528} C_VEL
LIN {X 0,Y 594.446,Z 355.817,A -85,B 0,C 180,E1 -1250.215,E2 -1250.215} C_VEL
LIN {X 0,Y 594.404,Z 365.592,A -85,B 0,C 180,E1 -1250.987,E2 -1250.987} C_VEL
LIN {X 0,Y 594.366,Z 374.486,A -85,B 0,C 180,E1 -1251.843,E2 -1251.843} C_VEL
LIN {X 0,Y 594.345,Z 383.172,A -85,B 0,C 180,E1 -1252.868,E2 -1252.868} C_VEL
LIN {X 0,Y 594.29,Z 390.1,A -85,B 0,C 180,E1 -1253.89,E2 -1253.89} C_VEL
LIN {X 0,Y 594.254,Z 395.652,A -85,B 0,C 180,E1 -1254.911,E2 -1254.911} C_VEL
LIN {X 0,Y 594.263,Z 400.014,A -85,B 0,C 180,E1 -1255.931,E2 -1255.931} C_VEL
LIN {X 0,Y 594.268,Z 402.317,A -85,B 0,C 180,E1 -1256.61,E2 -1256.61} C_VEL
LIN {X 0,Y 594.225,Z 404.194,A -85,B 0,C 180,E1 -1257.288,E2 -1257.288} C_VEL
LIN {X 0,Y 594.24,Z 405.627,A -85,B 0,C 180,E1 -1257.967,E2 -1257.967} C_VEL
LIN {X 0,Y 594.241,Z 407.253,A -85,B 0,C 180,E1 -1259.322,E2 -1259.322} C_VEL
LIN {X 0,Y 594.236,Z 407.496,A -85,B 0,C 180,E1 -1260,E2 -1260} C_VEL
LIN {X 0,Y 594.239,Z 407.315,A -85,B 0,C 180,E1 -1260.678,E2 -1260.678} C_VEL
LIN {X 0,Y 594.239,Z 405.776,A -85,B 0,C 180,E1 -1262.033,E2 -1262.033} C_VEL
LIN {X 0,Y 594.226,Z 404.415,A -85,B 0,C 180,E1 -1262.712,E2 -1262.712} C_VEL
LIN {X 0,Y 594.289,Z 401.538,A -85,B 0,C 180,E1 -1263.729,E2 -1263.729} C_VEL
LIN {X 0,Y 594.241,Z 397.638,A -85,B 0,C 180,E1 -1264.749,E2 -1264.749} C_VEL
LIN {X 0,Y 594.299,Z 392.607,A -85,B 0,C 180,E1 -1265.769,E2 -1265.769} C_VEL
LIN {X 0,Y 594.316,Z 386.287,A -85,B 0,C 180,E1 -1266.791,E2 -1266.791} C_VEL
LIN {X 0,Y 594.346,Z 378.369,A -85,B 0,C 180,E1 -1267.816,E2 -1267.816} C_VEL
LIN {X 0,Y 594.381,Z 368.522,A -85,B 0,C 180,E1 -1268.842,E2 -1268.842} C_VEL
LIN {X 0,Y 594.428,Z 358.2,A -85,B 0,C 180,E1 -1269.7,E2 -1269.7} C_VEL
LIN {X 0,Y 594.506,Z 346.577,A -85,B 0,C 180,E1 -1270.472,E2 -1270.472} C_VEL
LIN {X 0,Y 594.559,Z 334.806,A -85,B 0,C 180,E1 -1271.083,E2 -1271.083} C_VEL
LIN {X 0,Y 594.6,Z 321.726,A -85,B 0,C 180,E1 -1271.592,E2 -1271.592} C_VEL
LIN {X 0,Y 594.661,Z 314.226,A -85,B 0,C 180,E1 -1271.814,E2 -1271.814} C_VEL
LIN {X 0,Y 594.272,Z 310.901,A -85,B 0,C 180,E1 -1271.97,E2 -1271.97} C_VEL
LIN {X 0,Y 593.364,Z 308.226,A -85,B 0,C 180,E1 -1272.212,E2 -1272.212} C_VEL
LIN {X 0,Y 591.519,Z 305.316,A -85,B 0,C 180,E1 -1272.67,E2 -1272.67} C_VEL
LIN {X 0,Y 589.507,Z 303.493,A -85,B 0,C 180,E1 -1273.214,E2 -1273.214} C_VEL
LIN {X 0,Y 587.473,Z 302.035,A -85,B 0,C 180,E1 -1274.008,E2 -1274.008} C_VEL
LIN {X 0,Y 587.136,Z 301.498,A -85,B 0,C 180,E1 -1274.419,E2 -1274.419} C_VEL
LIN {X 0,Y 587.147,Z 298.549,A -85,B 0,C 180,E1 -1276.747,E2 -1276.747} C_VEL
LIN {X 0,Y 587.116,Z 295.009,A -85,B 0,C 180,E1 -1279.583,E2 -1279.583} C_VEL
LIN {X 0,Y 587.139,Z 292.304,A -85,B 0,C 180,E1 -1281.782,E2 -1281.782} C_VEL
LIN {X 0,Y 587.179,Z 288.782,A -85,B 0,C 180,E1 -1284.766,E2 -1284.766} C_VEL
LIN {X 0,Y 587.206,Z 285.799,A -85,B 0,C 180,E1 -1287.665,E2 -1287.665} C_VEL
LIN {X 0,Y 587.204,Z 282.575,A -85,B 0,C 180,E1 -1290.487,E2 -1290.487} C_VEL
LIN {X 0,Y 587.193,Z 279.321,A -85,B 0,C 180,E1 -1293.406,E2 -1293.406} C_VEL
LIN {X 0,Y 587.219,Z 278.28,A -85,B 0,C 180,E1 -1294.329,E2 -1294.329} C_VEL
LIN {X 0,Y 587.276,Z 277.954,A -85,B 0,C 180,E1 -1295.901,E2 -1295.901} C_VEL
LIN {X 0,Y 587.335,Z 277.947,A -85,B 0,C 180,E1 -1298.479,E2 -1298.479} C_VEL
LIN {X 0,Y 587.337,Z 277.947,A -85,B 0,C 180,E1 -1301.157,E2 -1301.157} C_VEL
LIN {X 0,Y 587.314,Z 277.952,A -85,B 0,C 180,E1 -1304.112,E2 -1304.112} C_VEL
LIN {X 0,Y 587.293,Z 277.951,A -85,B 0,C 180,E1 -1306.991,E2 -1306.991} C_VEL
LIN {X 0,Y 587.259,Z 277.962,A -85,B 0,C 180,E1 -1309.64,E2 -1309.64} C_VEL
LIN {X 0,Y 587.308,Z 282.231,A -85,B 0,C 180,E1 -1312.166,E2 -1312.166} C_VEL
LIN {X 0,Y 587.239,Z 286.364,A -85,B 0,C 180,E1 -1314.938,E2 -1314.938} C_VEL
LIN {X 0,Y 587.243,Z 290.001,A -85,B 0,C 180,E1 -1317.415,E2 -1317.415} C_VEL
LIN {X 0,Y 587.237,Z 293.523,A -85,B 0,C 180,E1 -1319.824,E2 -1319.824} C_VEL
LIN {X 0,Y 587.201,Z 297.281,A -85,B 0,C 180,E1 -1322.335,E2 -1322.335} C_VEL
LIN {X 0,Y 587.186,Z 300.66,A -85,B 0,C 180,E1 -1324.476,E2 -1324.476} C_VEL
LIN {X 0,Y 587.2,Z 305.501,A -85,B 0,C 180,E1 -1327.48,E2 -1327.48} C_VEL
LIN {X 0,Y 587.15,Z 310.342,A -85,B 0,C 180,E1 -1330.418,E2 -1330.418} C_VEL
LIN {X 0,Y 587.162,Z 314.601,A -85,B 0,C 180,E1 -1332.893,E2 -1332.893} C_VEL
LIN {X 0,Y 588.314,Z 320.393,A -85,B 0,C 180,E1 -1333.015,E2 -1333.015} C_VEL
LIN {X 0,Y 588.238,Z 334.96,A -85,B 0,C 180,E1 -1333.314,E2 -1333.314} C_VEL
LIN {X 0,Y 588.086,Z 350.525,A -85,B 0,C 180,E1 -1333.779,E2 -1333.779} C_VEL
LIN {X 0,Y 588.006,Z 363.789,A -85,B 0,C 180,E1 -1334.311,E2 -1334.311} C_VEL
LIN {X 0,Y 587.836,Z 377.86,A -85,B 0,C 180,E1 -1335.016,E2 -1335.016} C_VEL
LIN {X 0,Y 587.723,Z 391.197,A -85,B 0,C 180,E1 -1335.84,E2 -1335.84} C_VEL
LIN {X 0,Y 587.582,Z 404.745,A -85,B 0,C 180,E1 -1336.864,E2 -1336.864} C_VEL
LIN {X 0,Y 587.454,Z 416.272,A -85,B 0,C 180,E1 -1337.915,E2 -1337.915} C_VEL
LIN {X 0,Y 587.351,Z 426.013,A -85,B 0,C 180,E1 -1338.962,E2 -1338.962} C_VEL
LIN {X 0,Y 587.311,Z 435.544,A -85,B 0,C 180,E1 -1340.182,E2 -1340.182} C_VEL
LIN {X 0,Y 587.268,Z 443.458,A -85,B 0,C 180,E1 -1341.397,E2 -1341.397} C_VEL
LIN {X 0,Y 587.216,Z 450.881,A -85,B 0,C 180,E1 -1342.781,E2 -1342.781} C_VEL
LIN {X 0,Y 587.227,Z 456.772,A -85,B 0,C 180,E1 -1344.161,E2 -1344.161} C_VEL
LIN {X 0,Y 587.134,Z 460.249,A -85,B 0,C 180,E1 -1345.193,E2 -1345.193} C_VEL
LIN {X 0,Y 587.179,Z 463.8,A -85,B 0,C 180,E1 -1346.569,E2 -1346.569} C_VEL
LIN {X 0,Y 587.14,Z 466.136,A -85,B 0,C 180,E1 -1347.942,E2 -1347.942} C_VEL
LIN {X 0,Y 587.135,Z 467.318,A -85,B 0,C 180,E1 -1349.314,E2 -1349.314} C_VEL
LIN {X 0,Y 587.136,Z 467.35,A -85,B 0,C 180,E1 -1350.686,E2 -1350.686} C_VEL
LIN {X 0,Y 587.14,Z 466.239,A -85,B 0,C 180,E1 -1352.058,E2 -1352.058} C_VEL
LIN {X 0,Y 587.181,Z 463.989,A -85,B 0,C 180,E1 -1353.431,E2 -1353.431} C_VEL
LIN {X 0,Y 587.134,Z 460.527,A -85,B 0,C 180,E1 -1354.806,E2 -1354.806} C_VEL
LIN {X 0,Y 587.183,Z 455.779,A -85,B 0,C 180,E1 -1356.184,E2 -1356.184} C_VEL
LIN {X 0,Y 587.229,Z 449.643,A -85,B 0,C 180,E1 -1357.565,E2 -1357.565} C_VEL
LIN {X 0,Y 587.266,Z 441.948,A -85,B 0,C 180,E1 -1358.95,E2 -1358.95} C_VEL
LIN {X 0,Y 587.351,Z 433.701,A -85,B 0,C 180,E1 -1360.165,E2 -1360.165} C_VEL
LIN {X 0,Y 587.376,Z 423.764,A -85,B 0,C 180,E1 -1361.386,E2 -1361.386} C_VEL
LIN {X 0,Y 587.498,Z 413.627,A -85,B 0,C 180,E1 -1362.435,E2 -1362.435} C_VEL
LIN {X 0,Y 587.62,Z 401.587,A -85,B 0,C 180,E1 -1363.487,E2 -1363.487} C_VEL
LIN {X 0,Y 587.75,Z 388.864,A -85,B 0,C 180,E1 -1364.406,E2 -1364.406} C_VEL
LIN {X 0,Y 587.89,Z 376.298,A -85,B 0,C 180,E1 -1365.159,E2 -1365.159} C_VEL
LIN {X 0,Y 587.968,Z 363.82,A -85,B 0,C 180,E1 -1365.779,E2 -1365.779} C_VEL
LIN {X 0,Y 588.137,Z 349.265,A -85,B 0,C 180,E1 -1366.353,E2 -1366.353} C_VEL
LIN {X 0,Y 588.232,Z 333.525,A -85,B 0,C 180,E1 -1366.811,E2 -1366.811} C_VEL
LIN {X 0,Y 588.231,Z 319.244,A -85,B 0,C 180,E1 -1367.096,E2 -1367.096} C_VEL
LIN {X 0,Y 587.163,Z 314.474,A -85,B 0,C 180,E1 -1367.204,E2 -1367.204} C_VEL
LIN {X 0,Y 587.15,Z 310.492,A -85,B 0,C 180,E1 -1369.582,E2 -1369.582} C_VEL
LIN {X 0,Y 587.199,Z 305.648,A -85,B 0,C 180,E1 -1372.519,E2 -1372.519} C_VEL
LIN {X 0,Y 587.185,Z 300.804,A -85,B 0,C 180,E1 -1375.524,E2 -1375.524} C_VEL
LIN {X 0,Y 587.218,Z 297.171,A -85,B 0,C 180,E1 -1377.824,E2 -1377.824} C_VEL
LIN {X 0,Y 587.241,Z 293.189,A -85,B 0,C 180,E1 -1380.494,E2 -1380.494} C_VEL
LIN {X 0,Y 587.244,Z 289.397,A -85,B 0,C 180,E1 -1383.097,E2 -1383.097} C_VEL
LIN {X 0,Y 587.276,Z 285.25,A -85,B 0,C 180,E1 -1385.901,E2 -1385.901} C_VEL
LIN {X 0,Y 587.312,Z 281.362,A -85,B 0,C 180,E1 -1388.481,E2 -1388.481} C_VEL
LIN {X 0,Y 587.258,Z 277.963,A -85,B 0,C 180,E1 -1390.484,E2 -1390.484} C_VEL
LIN {X 0,Y 587.313,Z 277.951,A -85,B 0,C 180,E1 -1393.118,E2 -1393.118} C_VEL
LIN {X 0,Y 587.314,Z 277.949,A -85,B 0,C 180,E1 -1396.048,E2 -1396.048} C_VEL
LIN {X 0,Y 587.332,Z 277.95,A -85,B 0,C 180,E1 -1398.925,E2 -1398.925} C_VEL
LIN {X 0,Y 587.311,Z 277.951,A -85,B 0,C 180,E1 -1401.519,E2 -1401.519} C_VEL
LIN {X 0,Y 587.33,Z 277.947,A -85,B 0,C 180,E1 -1404.458,E2 -1404.458} C_VEL
LIN {X 0,Y 587.339,Z 277.952,A -85,B 0,C 180,E1 -1406.888,E2 -1406.888} C_VEL
LIN {X 0,Y 587.33,Z 277.948,A -85,B 0,C 180,E1 -1409.83,E2 -1409.83} C_VEL
LIN {X 0,Y 587.295,Z 277.951,A -85,B 0,C 180,E1 -1412.952,E2 -1412.952} C_VEL
LIN {X 0,Y 587.353,Z 277.949,A -85,B 0,C 180,E1 -1415.42,E2 -1415.42} C_VEL
LIN {X 0,Y 587.323,Z 277.949,A -85,B 0,C 180,E1 -1418.226,E2 -1418.226} C_VEL
LIN {X 0,Y 587.33,Z 277.947,A -85,B 0,C 180,E1 -1421.15,E2 -1421.15} C_VEL
LIN {X 0,Y 587.301,Z 277.952,A -85,B 0,C 180,E1 -1424.024,E2 -1424.024} C_VEL
LIN {X 0,Y 587.357,Z 277.943,A -85,B 0,C 180,E1 -1426.154,E2 -1426.154} C_VEL
LIN {X 0,Y 587.339,Z 277.947,A -85,B 0,C 180,E1 -1428.962,E2 -1428.962} C_VEL
LIN {X 0,Y 587.338,Z 277.951,A -85,B 0,C 180,E1 -1431.744,E2 -1431.744} C_VEL
LIN {X 0,Y 587.327,Z 277.946,A -85,B 0,C 180,E1 -1434.507,E2 -1434.507} C_VEL
LIN {X 0,Y 587.378,Z 277.943,A -85,B 0,C 180,E1 -1437.257,E2 -1437.257} C_VEL
LIN {X 0,Y 587.385,Z 277.942,A -85,B 0,C 180,E1 -1440,E2 -1440} C_VEL
LIN {X 0,Y 587.349,Z 277.944,A -85,B 0,C 180,E1 -1442.743,E2 -1442.743} C_VEL
LIN {X 0,Y 587.352,Z 277.947,A -85,B 0,C 180,E1 -1445.493,E2 -1445.493} C_VEL
LIN {X 0,Y 587.333,Z 277.949,A -85,B 0,C 180,E1 -1448.256,E2 -1448.256} C_VEL
LIN {X 0,Y 587.35,Z 277.943,A -85,B 0,C 180,E1 -1451.134,E2 -1451.134} C_VEL
LIN {X 0,Y 587.328,Z 277.951,A -85,B 0,C 180,E1 -1453.846,E2 -1453.846} C_VEL
LIN {X 0,Y 587.33,Z 277.951,A -85,B 0,C 180,E1 -1456.808,E2 -1456.808} C_VEL
LIN {X 0,Y 587.344,Z 277.945,A -85,B 0,C 180,E1 -1459.575,E2 -1459.575} C_VEL
LIN {X 0,Y 587.337,Z 277.946,A -85,B 0,C 180,E1 -1462.514,E2 -1462.514} C_VEL
LIN {X 0,Y 587.308,Z 277.952,A -85,B 0,C 180,E1 -1465.518,E2 -1465.518} C_VEL
LIN {X 0,Y 587.305,Z 277.95,A -85,B 0,C 180,E1 -1467.82,E2 -1467.82} C_VEL
LIN {X 0,Y 587.34,Z 277.949,A -85,B 0,C 180,E1 -1470.51,E2 -1470.51} C_VEL
LIN {X 0,Y 587.334,Z 277.951,A -85,B 0,C 180,E1 -1473.397,E2 -1473.397} C_VEL
LIN {X 0,Y 587.283,Z 277.953,A -85,B 0,C 180,E1 -1475.901,E2 -1475.901} C_VEL
LIN {X 0,Y 587.312,Z 277.956,A -85,B 0,C 180,E1 -1478.481,E2 -1478.481} C_VEL
LIN {X 0,Y 587.335,Z 277.946,A -85,B 0,C 180,E1 -1481.157,E2 -1481.157} C_VEL
LIN {X 0,Y 587.311,Z 277.95,A -85,B 0,C 180,E1 -1484.112,E2 -1484.112} C_VEL
LIN {X 0,Y 587.292,Z 277.957,A -85,B 0,C 180,E1 -1486.992,E2 -1486.992} C_VEL
LIN {X 0,Y 587.304,Z 277.952,A -85,B 0,C 180,E1 -1489.745,E2 -1489.745} C_VEL
LIN {X 0,Y 587.346,Z 277.949,A -85,B 0,C 180,E1 -1492.393,E2 -1492.393} C_VEL
LIN {X 0,Y 587.357,Z 278.021,A -85,B 0,C 180,E1 -1494.903,E2 -1494.903} C_VEL
LIN {X 0,Y 588.756,Z 284.563,A -85,B 0,C 180,E1 -1496.079,E2 -1496.079} C_VEL
LIN {X 0,Y 588.41,Z 302.161,A -85,B 0,C 180,E1 -1498.897,E2 -1498.897} C_VEL
LIN {X 0,Y 588.262,Z 318.893,A -85,B 0,C 180,E1 -1501.453,E2 -1501.453} C_VEL
LIN {X 0,Y 588.094,Z 338.086,A -85,B 0,C 180,E1 -1504.329,E2 -1504.329} C_VEL
LIN {X 0,Y 587.867,Z 358.091,A -85,B 0,C 180,E1 -1507.254,E2 -1507.254} C_VEL
LIN {X 0,Y 587.724,Z 379.031,A -85,B 0,C 180,E1 -1510.256,E2 -1510.256} C_VEL
LIN {X 0,Y 587.565,Z 396.867,A -85,B 0,C 180,E1 -1512.763,E2 -1512.763} C_VEL
LIN {X 0,Y 588.32,Z 401.012,A -85,B 0,C 180,E1 -1512.838,E2 -1512.838} C_VEL
LIN {X 0,Y 588.251,Z 416.995,A -85,B 0,C 180,E1 -1513.088,E2 -1513.088} C_VEL
LIN {X 0,Y 588.166,Z 432.29,A -85,B 0,C 180,E1 -1513.469,E2 -1513.469} C_VEL
LIN {X 0,Y 588.06,Z 446.434,A -85,B 0,C 180,E1 -1513.956,E2 -1513.956} C_VEL
LIN {X 0,Y 587.938,Z 460.373,A -85,B 0,C 180,E1 -1514.576,E2 -1514.576} C_VEL
LIN {X 0,Y 587.832,Z 473.212,A -85,B 0,C 180,E1 -1515.282,E2 -1515.282} C_VEL
LIN {X 0,Y 587.675,Z 486.369,A -85,B 0,C 180,E1 -1516.162,E2 -1516.162} C_VEL
LIN {X 0,Y 587.558,Z 497.387,A -85,B 0,C 180,E1 -1517.04,E2 -1517.04} C_VEL
LIN {X 0,Y 587.446,Z 508.51,A -85,B 0,C 180,E1 -1518.09,E2 -1518.09} C_VEL
LIN {X 0,Y 587.384,Z 519.303,A -85,B 0,C 180,E1 -1519.312,E2 -1519.312} C_VEL
LIN {X 0,Y 587.276,Z 528.293,A -85,B 0,C 180,E1 -1520.529,E2 -1520.529} C_VEL
LIN {X 0,Y 587.255,Z 535.752,A -85,B 0,C 180,E1 -1521.743,E2 -1521.743} C_VEL
LIN {X 0,Y 587.206,Z 542.703,A -85,B 0,C 180,E1 -1523.126,E2 -1523.126} C_VEL
LIN {X 0,Y 587.199,Z 548.161,A -85,B 0,C 180,E1 -1524.506,E2 -1524.506} C_VEL
LIN {X 0,Y 587.167,Z 552.289,A -85,B 0,C 180,E1 -1525.882,E2 -1525.882} C_VEL
LIN {X 0,Y 587.129,Z 555.187,A -85,B 0,C 180,E1 -1527.256,E2 -1527.256} C_VEL
LIN {X 0,Y 587.145,Z 556.912,A -85,B 0,C 180,E1 -1528.628,E2 -1528.628} C_VEL
LIN {X 0,Y 587.134,Z 557.5,A -85,B 0,C 180,E1 -1530,E2 -1530} C_VEL
LIN {X 0,Y 587.145,Z 556.912,A -85,B 0,C 180,E1 -1531.372,E2 -1531.372} C_VEL
LIN {X 0,Y 587.129,Z 555.185,A -85,B 0,C 180,E1 -1532.745,E2 -1532.745} C_VEL
LIN {X 0,Y 587.167,Z 552.288,A -85,B 0,C 180,E1 -1534.118,E2 -1534.118} C_VEL
LIN {X 0,Y 587.199,Z 548.162,A -85,B 0,C 180,E1 -1535.495,E2 -1535.495} C_VEL
LIN {X 0,Y 587.206,Z 542.702,A -85,B 0,C 180,E1 -1536.874,E2 -1536.874} C_VEL
LIN {X 0,Y 587.255,Z 535.749,A -85,B 0,C 180,E1 -1538.257,E2 -1538.257} C_VEL
LIN {X 0,Y 587.286,Z 527.089,A -85,B 0,C 180,E1 -1539.645,E2 -1539.645} C_VEL
LIN {X 0,Y 587.371,Z 517.875,A -85,B 0,C 180,E1 -1540.863,E2 -1540.863} C_VEL
LIN {X 0,Y 587.446,Z 508.507,A -85,B 0,C 180,E1 -1541.91,E2 -1541.91} C_VEL
LIN {X 0,Y 587.558,Z 497.385,A -85,B 0,C 180,E1 -1542.96,E2 -1542.96} C_VEL
LIN {X 0,Y 587.711,Z 484.815,A -85,B 0,C 180,E1 -1543.953,E2 -1543.953} C_VEL
LIN {X 0,Y 587.833,Z 471.778,A -85,B 0,C 180,E1 -1544.807,E2 -1544.807} C_VEL
LIN {X 0,Y 587.951,Z 458.602,A -85,B 0,C 180,E1 -1545.513,E2 -1545.513} C_VEL
LIN {X 0,Y 588.094,Z 444.176,A -85,B 0,C 180,E1 -1546.132,E2 -1546.132} C_VEL
LIN {X 0,Y 588.196,Z 429.245,A -85,B 0,C 180,E1 -1546.62,E2 -1546.62} C_VEL
LIN {X 0,Y 588.253,Z 414.286,A -85,B 0,C 180,E1 -1546.965,E2 -1546.965} C_VEL
LIN {X 0,Y 588.276,Z 400.498,A -85,B 0,C 180,E1 -1547.17,E2 -1547.17} C_VEL
LIN {X 0,Y 587.576,Z 396.746,A -85,B 0,C 180,E1 -1547.247,E2 -1547.247} C_VEL
LIN {X 0,Y 587.738,Z 375.19,A -85,B 0,C 180,E1 -1550.29,E2 -1550.29} C_VEL
LIN {X 0,Y 587.914,Z 354.718,A -85,B 0,C 180,E1 -1553.234,E2 -1553.234} C_VEL
LIN {X 0,Y 588.086,Z 335.525,A -85,B 0,C 180,E1 -1556.052,E2 -1556.052} C_VEL
LIN {X 0,Y 588.298,Z 317.611,A -85,B 0,C 180,E1 -1558.74,E2 -1558.74} C_VEL
LIN {X 0,Y 588.5,Z 301.127,A -85,B 0,C 180,E1 -1561.298,E2 -1561.298} C_VEL
LIN {X 0,Y 588.874,Z 287.777,A -85,B 0,C 180,E1 -1563.503,E2 -1563.503} C_VEL
LIN {X 0,Y 589,Z 284.394,A -85,B 0,C 180,E1 -1564.112,E2 -1564.112} C_VEL
LIN {X 0,Y 587.314,Z 277.954,A -85,B 0,C 180,E1 -1565.56,E2 -1565.56} C_VEL
LIN {X 0,Y 587.324,Z 277.955,A -85,B 0,C 180,E1 -1568.48,E2 -1568.48} C_VEL
LIN {X 0,Y 587.334,Z 277.953,A -85,B 0,C 180,E1 -1571.157,E2 -1571.157} C_VEL
LIN {X 0,Y 587.322,Z 277.954,A -85,B 0,C 180,E1 -1574.113,E2 -1574.113} C_VEL
LIN {X 0,Y 587.317,Z 277.953,A -85,B 0,C 180,E1 -1576.994,E2 -1576.994} C_VEL
LIN {X 0,Y 587.307,Z 277.954,A -85,B 0,C 180,E1 -1579.745,E2 -1579.745} C_VEL
LIN {X 0,Y 587.346,Z 277.95,A -85,B 0,C 180,E1 -1582.393,E2 -1582.393} C_VEL
LIN {X 0,Y 587.265,Z 277.962,A -85,B 0,C 180,E1 -1584.467,E2 -1584.467} C_VEL
LIN {X 0,Y 587.329,Z 280.922,A -85,B 0,C 180,E1 -1586.89,E2 -1586.89} C_VEL
LIN {X 0,Y 587.321,Z 283.751,A -85,B 0,C 180,E1 -1589.493,E2 -1589.493} C_VEL
LIN {X 0,Y 587.303,Z 286.399,A -85,B 0,C 180,E1 -1592.18,E2 -1592.18} C_VEL
LIN {X 0,Y 587.234,Z 288.293,A -85,B 0,C 180,E1 -1594.479,E2 -1594.479} C_VEL
LIN {X 0,Y 587.184,Z 289.525,A -85,B 0,C 180,E1 -1595.987,E2 -1595.987} C_VEL
LIN {X 0,Y 587.178,Z 293.151,A -85,B 0,C 180,E1 -1599.002,E2 -1599.002} C_VEL
LIN {X 0,Y 587.126,Z 296.7,A -85,B 0,C 180,E1 -1601.867,E2 -1601.867} C_VEL
LIN {X 0,Y 587.152,Z 299.403,A -85,B 0,C 180,E1 -1604.02,E2 -1604.02} C_VEL
LIN {X 0,Y 587.139,Z 303.008,A -85,B 0,C 180,E1 -1606.854,E2 -1606.854} C_VEL
LIN {X 0,Y 587.173,Z 304.532,A -85,B 0,C 180,E1 -1607.909,E2 -1607.909} C_VEL
LIN {X 0,Y 587.699,Z 309.893,A -85,B 0,C 180,E1 -1608.03,E2 -1608.03} C_VEL
LIN {X 0,Y 587.628,Z 323.185,A -85,B 0,C 180,E1 -1608.408,E2 -1608.408} C_VEL
LIN {X 0,Y 587.6,Z 335.704,A -85,B 0,C 180,E1 -1608.915,E2 -1608.915} C_VEL
LIN {X 0,Y 587.489,Z 347.945,A -85,B 0,C 180,E1 -1609.576,E2 -1609.576} C_VEL
LIN {X 0,Y 587.393,Z 359.318,A -85,B 0,C 180,E1 -1610.357,E2 -1610.357} C_VEL
LIN {X 0,Y 587.337,Z 369.375,A -85,B 0,C 180,E1 -1611.224,E2 -1611.224} C_VEL
LIN {X 0,Y 587.274,Z 379.078,A -85,B 0,C 180,E1 -1612.263,E2 -1612.263} C_VEL
LIN {X 0,Y 587.236,Z 385.648,A -85,B 0,C 180,E1 -1613.126,E2 -1613.126} C_VEL
LIN {X 0,Y 587.237,Z 392.118,A -85,B 0,C 180,E1 -1614.161,E2 -1614.161} C_VEL
LIN {X 0,Y 587.146,Z 397.258,A -85,B 0,C 180,E1 -1615.194,E2 -1615.194} C_VEL
LIN {X 0,Y 587.213,Z 401.248,A -85,B 0,C 180,E1 -1616.226,E2 -1616.226} C_VEL
LIN {X 0,Y 587.132,Z 404.196,A -85,B 0,C 180,E1 -1617.256,E2 -1617.256} C_VEL
LIN {X 0,Y 587.139,Z 405.627,A -85,B 0,C 180,E1 -1617.942,E2 -1617.942} C_VEL
LIN {X 0,Y 587.141,Z 407.254,A -85,B 0,C 180,E1 -1619.314,E2 -1619.314} C_VEL
LIN {X 0,Y 587.137,Z 407.496,A -85,B 0,C 180,E1 -1620,E2 -1620} C_VEL
LIN {X 0,Y 587.14,Z 407.315,A -85,B 0,C 180,E1 -1620.686,E2 -1620.686} C_VEL
LIN {X 0,Y 587.138,Z 405.775,A -85,B 0,C 180,E1 -1622.058,E2 -1622.058} C_VEL
LIN {X 0,Y 587.133,Z 404.414,A -85,B 0,C 180,E1 -1622.744,E2 -1622.744} C_VEL
LIN {X 0,Y 587.213,Z 401.536,A -85,B 0,C 180,E1 -1623.774,E2 -1623.774} C_VEL
LIN {X 0,Y 587.147,Z 397.635,A -85,B 0,C 180,E1 -1624.806,E2 -1624.806} C_VEL
LIN {X 0,Y 587.229,Z 392.605,A -85,B 0,C 180,E1 -1625.839,E2 -1625.839} C_VEL
LIN {X 0,Y 587.23,Z 386.283,A -85,B 0,C 180,E1 -1626.874,E2 -1626.874} C_VEL
LIN {X 0,Y 587.288,Z 378.365,A -85,B 0,C 180,E1 -1627.91,E2 -1627.91} C_VEL
LIN {X 0,Y 587.343,Z 368.516,A -85,B 0,C 180,E1 -1628.949,E2 -1628.949} C_VEL
LIN {X 0,Y 587.413,Z 358.193,A -85,B 0,C 180,E1 -1629.816,E2 -1629.816} C_VEL
LIN {X 0,Y 587.51,Z 346.566,A -85,B 0,C 180,E1 -1630.598,E2 -1630.598} C_VEL
LIN {X 0,Y 587.59,Z 335.627,A -85,B 0,C 180,E1 -1631.179,E2 -1631.179} C_VEL
LIN {X 0,Y 587.627,Z 322.949,A -85,B 0,C 180,E1 -1631.689,E2 -1631.689} C_VEL
LIN {X 0,Y 587.703,Z 309.983,A -85,B 0,C 180,E1 -1632.058,E2 -1632.058} C_VEL
LIN {X 0,Y 587.141,Z 304.334,A -85,B 0,C 180,E1 -1632.201,E2 -1632.201} C_VEL
LIN {X 0,Y 587.136,Z 301.498,A -85,B 0,C 180,E1 -1634.419,E2 -1634.419} C_VEL
LIN {X 0,Y 586.448,Z 300.798,A -85,B 0,C 180,E1 -1634.987,E2 -1634.987} C_VEL
LIN {X 0,Y 583.559,Z 299.73,A -85,B 0,C 180,E1 -1635.911,E2 -1635.911} C_VEL
LIN {X 0,Y 581.135,Z 298.887,A -85,B 0,C 180,E1 -1636.654,E2 -1636.654} C_VEL
LIN {X 0,Y 580.107,Z 298.212,A -85,B 0,C 180,E1 -1637.227,E2 -1637.227} C_VEL
LIN {X 0,Y 580.03,Z 297.975,A -85,B 0,C 180,E1 -1637.421,E2 -1637.421} C_VEL
LIN {X 0,Y 580.052,Z 295.008,A -85,B 0,C 180,E1 -1639.831,E2 -1639.831} C_VEL
LIN {X 0,Y 580.042,Z 292.303,A -85,B 0,C 180,E1 -1642.062,E2 -1642.062} C_VEL
LIN {X 0,Y 580.11,Z 289.463,A -85,B 0,C 180,E1 -1644.684,E2 -1644.684} C_VEL
LIN {X 0,Y 580.132,Z 286.665,A -85,B 0,C 180,E1 -1647.41,E2 -1647.41} C_VEL
LIN {X 0,Y 580.146,Z 283.971,A -85,B 0,C 180,E1 -1649.781,E2 -1649.781} C_VEL
LIN {X 0,Y 580.112,Z 281.27,A -85,B 0,C 180,E1 -1652.212,E2 -1652.212} C_VEL
LIN {X 0,Y 580.154,Z 278.847,A -85,B 0,C 180,E1 -1654.537,E2 -1654.537} C_VEL
LIN {X 0,Y 580.302,Z 278.828,A -85,B 0,C 180,E1 -1657.268,E2 -1657.268} C_VEL
LIN {X 0,Y 580.299,Z 278.823,A -85,B 0,C 180,E1 -1660.271,E2 -1660.271} C_VEL
LIN {X 0,Y 580.279,Z 278.83,A -85,B 0,C 180,E1 -1662.706,E2 -1662.706} C_VEL
LIN {X 0,Y 580.253,Z 278.828,A -85,B 0,C 180,E1 -1665.611,E2 -1665.611} C_VEL
LIN {X 0,Y 580.247,Z 278.834,A -85,B 0,C 180,E1 -1668.228,E2 -1668.228} C_VEL
LIN {X 0,Y 580.223,Z 278.939,A -85,B 0,C 180,E1 -1669.738,E2 -1669.738} C_VEL
LIN {X 0,Y 580.276,Z 282.694,A -85,B 0,C 180,E1 -1671.929,E2 -1671.929} C_VEL
LIN {X 0,Y 580.2,Z 286.485,A -85,B 0,C 180,E1 -1674.449,E2 -1674.449} C_VEL
LIN {X 0,Y 580.182,Z 290.124,A -85,B 0,C 180,E1 -1676.968,E2 -1676.968} C_VEL
LIN {X 0,Y 580.194,Z 293.707,A -85,B 0,C 180,E1 -1679.419,E2 -1679.419} C_VEL
LIN {X 0,Y 580.145,Z 297.657,A -85,B 0,C 180,E1 -1682.17,E2 -1682.17} C_VEL
LIN {X 0,Y 580.097,Z 301.871,A -85,B 0,C 180,E1 -1684.91,E2 -1684.91} C_VEL
LIN {X 0,Y 580.137,Z 305.502,A -85,B 0,C 180,E1 -1687.191,E2 -1687.191} C_VEL
LIN {X 0,Y 580.075,Z 310.343,A -85,B 0,C 180,E1 -1690.169,E2 -1690.169} C_VEL
LIN {X 0,Y 580.082,Z 314.479,A -85,B 0,C 180,E1 -1692.673,E2 -1692.673} C_VEL
LIN {X 0,Y 581.514,Z 321.549,A -85,B 0,C 180,E1 -1692.83,E2 -1692.83} C_VEL
LIN {X 0,Y 581.424,Z 336.75,A -85,B 0,C 180,E1 -1693.156,E2 -1693.156} C_VEL
LIN {X 0,Y 581.243,Z 351.8,A -85,B 0,C 180,E1 -1693.627,E2 -1693.627} C_VEL
LIN {X 0,Y 581.124,Z 365.733,A -85,B 0,C 180,E1 -1694.21,E2 -1694.21} C_VEL
LIN {X 0,Y 580.933,Z 379.435,A -85,B 0,C 180,E1 -1694.924,E2 -1694.924} C_VEL
LIN {X 0,Y 580.808,Z 392.89,A -85,B 0,C 180,E1 -1695.786,E2 -1695.786} C_VEL
LIN {X 0,Y 580.61,Z 404.754,A -85,B 0,C 180,E1 -1696.704,E2 -1696.704} C_VEL
LIN {X 0,Y 580.48,Z 416.273,A -85,B 0,C 180,E1 -1697.767,E2 -1697.767} C_VEL
LIN {X 0,Y 580.31,Z 427.082,A -85,B 0,C 180,E1 -1698.953,E2 -1698.953} C_VEL
LIN {X 0,Y 580.241,Z 436.788,A -85,B 0,C 180,E1 -1700.237,E2 -1700.237} C_VEL
LIN {X 0,Y 580.18,Z 444.47,A -85,B 0,C 180,E1 -1701.466,E2 -1701.466} C_VEL
LIN {X 0,Y 580.132,Z 450.885,A -85,B 0,C 180,E1 -1702.692,E2 -1702.692} C_VEL
LIN {X 0,Y 580.132,Z 456.777,A -85,B 0,C 180,E1 -1704.089,E2 -1704.089} C_VEL
LIN {X 0,Y 580.039,Z 460.252,A -85,B 0,C 180,E1 -1705.134,E2 -1705.134} C_VEL
LIN {X 0,Y 580.104,Z 463.804,A -85,B 0,C 180,E1 -1706.527,E2 -1706.527} C_VEL
LIN {X 0,Y 580.039,Z 466.135,A -85,B 0,C 180,E1 -1707.917,E2 -1707.917} C_VEL
LIN {X 0,Y 580.036,Z 467.312,A -85,B 0,C 180,E1 -1709.306,E2 -1709.306} C_VEL
LIN {X 0,Y 580.037,Z 467.344,A -85,B 0,C 180,E1 -1710.694,E2 -1710.694} C_VEL
LIN {X 0,Y 580.039,Z 466.237,A -85,B 0,C 180,E1 -1712.083,E2 -1712.083} C_VEL
LIN {X 0,Y 580.106,Z 463.991,A -85,B 0,C 180,E1 -1713.473,E2 -1713.473} C_VEL
LIN {X 0,Y 580.039,Z 460.527,A -85,B 0,C 180,E1 -1714.865,E2 -1714.865} C_VEL
LIN {X 0,Y 580.092,Z 455.772,A -85,B 0,C 180,E1 -1716.26,E2 -1716.26} C_VEL
LIN {X 0,Y 580.131,Z 451.303,A -85,B 0,C 180,E1 -1717.308,E2 -1717.308} C_VEL
LIN {X 0,Y 580.215,Z 443.979,A -85,B 0,C 180,E1 -1718.708,E2 -1718.708} C_VEL
LIN {X 0,Y 580.269,Z 436.186,A -85,B 0,C 180,E1 -1719.938,E2 -1719.938} C_VEL
LIN {X 0,Y 580.341,Z 426.464,A -85,B 0,C 180,E1 -1721.21,E2 -1721.21} C_VEL
LIN {X 0,Y 580.472,Z 417.177,A -85,B 0,C 180,E1 -1722.232,E2 -1722.232} C_VEL
LIN {X 0,Y 580.605,Z 406.833,A -85,B 0,C 180,E1 -1723.207,E2 -1723.207} C_VEL
LIN {X 0,Y 580.774,Z 395.561,A -85,B 0,C 180,E1 -1724.109,E2 -1724.109} C_VEL
LIN {X 0,Y 580.913,Z 382.516,A -85,B 0,C 180,E1 -1724.987,E2 -1724.987} C_VEL
LIN {X 0,Y 581.09,Z 369.527,A -85,B 0,C 180,E1 -1725.701,E2 -1725.701} C_VEL
LIN {X 0,Y 581.212,Z 355.266,A -85,B 0,C 180,E1 -1726.328,E2 -1726.328} C_VEL
LIN {X 0,Y 581.386,Z 340.776,A -85,B 0,C 180,E1 -1726.82,E2 -1726.82} C_VEL
LIN {X 0,Y 581.488,Z 325.006,A -85,B 0,C 180,E1 -1727.201,E2 -1727.201} C_VEL
LIN {X 0,Y 581.345,Z 320.187,A -85,B 0,C 180,E1 -1727.288,E2 -1727.288} C_VEL
LIN {X 0,Y 580.062,Z 314.473,A -85,B 0,C 180,E1 -1727.422,E2 -1727.422} C_VEL
LIN {X 0,Y 580.075,Z 310.491,A -85,B 0,C 180,E1 -1729.83,E2 -1729.83} C_VEL
LIN {X 0,Y 580.136,Z 305.647,A -85,B 0,C 180,E1 -1732.809,E2 -1732.809} C_VEL
LIN {X 0,Y 580.137,Z 300.803,A -85,B 0,C 180,E1 -1735.856,E2 -1735.856} C_VEL
LIN {X 0,Y 580.151,Z 297.266,A -85,B 0,C 180,E1 -1738.193,E2 -1738.193} C_VEL
LIN {X 0,Y 580.187,Z 293.698,A -85,B 0,C 180,E1 -1740.678,E2 -1740.678} C_VEL
LIN {X 0,Y 580.205,Z 289.88,A -85,B 0,C 180,E1 -1743.301,E2 -1743.301} C_VEL
LIN {X 0,Y 580.218,Z 286.319,A -85,B 0,C 180,E1 -1745.752,E2 -1745.752} C_VEL
LIN {X 0,Y 580.276,Z 282.731,A -85,B 0,C 180,E1 -1748.147,E2 -1748.147} C_VEL
LIN {X 0,Y 580.244,Z 278.836,A -85,B 0,C 180,E1 -1750.525,E2 -1750.525} C_VEL
LIN {X 0,Y 580.276,Z 278.83,A -85,B 0,C 180,E1 -1753.39,E2 -1753.39} C_VEL
LIN {X 0,Y 580.274,Z 278.827,A -85,B 0,C 180,E1 -1756.342,E2 -1756.342} C_VEL
LIN {X 0,Y 580.293,Z 278.825,A -85,B 0,C 180,E1 -1759.156,E2 -1759.156} C_VEL
LIN {X 0,Y 580.279,Z 278.832,A -85,B 0,C 180,E1 -1761.928,E2 -1761.928} C_VEL
LIN {X 0,Y 580.284,Z 278.825,A -85,B 0,C 180,E1 -1764.455,E2 -1764.455} C_VEL
LIN {X 0,Y 580.291,Z 278.83,A -85,B 0,C 180,E1 -1766.975,E2 -1766.975} C_VEL
LIN {X 0,Y 580.291,Z 278.823,A -85,B 0,C 180,E1 -1769.425,E2 -1769.425} C_VEL
LIN {X 0,Y 580.239,Z 278.834,A -85,B 0,C 180,E1 -1772.152,E2 -1772.152} C_VEL
LIN {X 0,Y 580.32,Z 278.827,A -85,B 0,C 180,E1 -1775.27,E2 -1775.27} C_VEL
LIN {X 0,Y 580.273,Z 278.825,A -85,B 0,C 180,E1 -1777.947,E2 -1777.947} C_VEL
LIN {X 0,Y 580.285,Z 278.825,A -85,B 0,C 180,E1 -1780.913,E2 -1780.913} C_VEL
LIN {X 0,Y 580.251,Z 278.832,A -85,B 0,C 180,E1 -1783.825,E2 -1783.825} C_VEL
LIN {X 0,Y 580.325,Z 278.82,A -85,B 0,C 180,E1 -1785.983,E2 -1785.983} C_VEL
LIN {X 0,Y 580.306,Z 278.825,A -85,B 0,C 180,E1 -1788.827,E2 -1788.827} C_VEL
LIN {X 0,Y 580.307,Z 278.825,A -85,B 0,C 180,E1 -1791.644,E2 -1791.644} C_VEL
LIN {X 0,Y 580.294,Z 278.822,A -85,B 0,C 180,E1 -1794.44,E2 -1794.44} C_VEL
LIN {X 0,Y 580.343,Z 278.82,A -85,B 0,C 180,E1 -1797.223,E2 -1797.223} C_VEL
LIN {X 0,Y 580.354,Z 278.817,A -85,B 0,C 180,E1 -1800,E2 -1800} C_VEL
LIN {X 0,Y 580.318,Z 278.82,A -85,B 0,C 180,E1 -1802.777,E2 -1802.777} C_VEL
LIN {X 0,Y 580.315,Z 278.822,A -85,B 0,C 180,E1 -1805.56,E2 -1805.56} C_VEL
LIN {X 0,Y 580.307,Z 278.826,A -85,B 0,C 180,E1 -1808.356,E2 -1808.356} C_VEL
LIN {X 0,Y 580.301,Z 278.82,A -85,B 0,C 180,E1 -1811.191,E2 -1811.191} C_VEL
LIN {X 0,Y 580.282,Z 278.826,A -85,B 0,C 180,E1 -1814.018,E2 -1814.018} C_VEL
LIN {X 0,Y 580.29,Z 278.829,A -85,B 0,C 180,E1 -1816.906,E2 -1816.906} C_VEL
LIN {X 0,Y 580.306,Z 278.824,A -85,B 0,C 180,E1 -1819.822,E2 -1819.822} C_VEL
LIN {X 0,Y 580.293,Z 278.823,A -85,B 0,C 180,E1 -1822.802,E2 -1822.802} C_VEL
LIN {X 0,Y 580.252,Z 278.828,A -85,B 0,C 180,E1 -1825.851,E2 -1825.851} C_VEL
LIN {X 0,Y 580.281,Z 278.827,A -85,B 0,C 180,E1 -1828.186,E2 -1828.186} C_VEL
LIN {X 0,Y 580.289,Z 278.826,A -85,B 0,C 180,E1 -1830.695,E2 -1830.695} C_VEL
LIN {X 0,Y 580.303,Z 278.826,A -85,B 0,C 180,E1 -1833.316,E2 -1833.316} C_VEL
LIN {X 0,Y 580.238,Z 278.831,A -85,B 0,C 180,E1 -1835.755,E2 -1835.755} C_VEL
LIN {X 0,Y 580.275,Z 278.828,A -85,B 0,C 180,E1 -1838.147,E2 -1838.147} C_VEL
LIN {X 0,Y 580.297,Z 278.823,A -85,B 0,C 180,E1 -1840.843,E2 -1840.843} C_VEL
LIN {X 0,Y 580.272,Z 278.831,A -85,B 0,C 180,E1 -1843.658,E2 -1843.658} C_VEL
LIN {X 0,Y 580.264,Z 278.83,A -85,B 0,C 180,E1 -1846.611,E2 -1846.611} C_VEL
LIN {X 0,Y 580.284,Z 278.827,A -85,B 0,C 180,E1 -1849.73,E2 -1849.73} C_VEL
LIN {X 0,Y 580.299,Z 278.827,A -85,B 0,C 180,E1 -1852.732,E2 -1852.732} C_VEL
LIN {X 0,Y 580.295,Z 278.901,A -85,B 0,C 180,E1 -1854.536,E2 -1854.536} C_VEL
LIN {X 0,Y 582.012,Z 285.92,A -85,B 0,C 180,E1 -1855.84,E2 -1855.84} C_VEL
LIN {X 0,Y 581.692,Z 302.093,A -85,B 0,C 180,E1 -1858.497,E2 -1858.497} C_VEL
LIN {X 0,Y 581.498,Z 318.893,A -85,B 0,C 180,E1 -1861.09,E2 -1861.09} C_VEL
LIN {X 0,Y 581.217,Z 338.141,A -85,B 0,C 180,E1 -1864.011,E2 -1864.011} C_VEL
LIN {X 0,Y 580.995,Z 357.131,A -85,B 0,C 180,E1 -1866.829,E2 -1866.829} C_VEL
LIN {X 0,Y 580.804,Z 376.472,A -85,B 0,C 180,E1 -1869.642,E2 -1869.642} C_VEL
LIN {X 0,Y 580.61,Z 396.982,A -85,B 0,C 180,E1 -1872.552,E2 -1872.552} C_VEL
LIN {X 0,Y 581.538,Z 402.441,A -85,B 0,C 180,E1 -1872.65,E2 -1872.65} C_VEL
LIN {X 0,Y 581.446,Z 418.754,A -85,B 0,C 180,E1 -1872.919,E2 -1872.919} C_VEL
LIN {X 0,Y 581.348,Z 433.809,A -85,B 0,C 180,E1 -1873.315,E2 -1873.315} C_VEL
LIN {X 0,Y 581.199,Z 448.678,A -85,B 0,C 180,E1 -1873.852,E2 -1873.852} C_VEL
LIN {X 0,Y 581.044,Z 462.123,A -85,B 0,C 180,E1 -1874.478,E2 -1874.478} C_VEL
LIN {X 0,Y 580.875,Z 476.042,A -85,B 0,C 180,E1 -1875.281,E2 -1875.281} C_VEL
LIN {X 0,Y 580.695,Z 488.698,A -85,B 0,C 180,E1 -1876.171,E2 -1876.171} C_VEL
LIN {X 0,Y 580.565,Z 499.338,A -85,B 0,C 180,E1 -1877.059,E2 -1877.059} C_VEL
LIN {X 0,Y 580.406,Z 510.141,A -85,B 0,C 180,E1 -1878.121,E2 -1878.121} C_VEL
LIN {X 0,Y 580.349,Z 520.759,A -85,B 0,C 180,E1 -1879.37,E2 -1879.37} C_VEL
LIN {X 0,Y 580.207,Z 529.416,A -85,B 0,C 180,E1 -1880.589,E2 -1880.589} C_VEL
LIN {X 0,Y 580.191,Z 535.752,A -85,B 0,C 180,E1 -1881.642,E2 -1881.642} C_VEL
LIN {X 0,Y 580.137,Z 542.703,A -85,B 0,C 180,E1 -1883.042,E2 -1883.042} C_VEL
LIN {X 0,Y 580.128,Z 548.161,A -85,B 0,C 180,E1 -1884.439,E2 -1884.439} C_VEL
LIN {X 0,Y 580.086,Z 552.289,A -85,B 0,C 180,E1 -1885.831,E2 -1885.831} C_VEL
LIN {X 0,Y 580.04,Z 555.187,A -85,B 0,C 180,E1 -1887.222,E2 -1887.222} C_VEL
LIN {X 0,Y 580.044,Z 556.912,A -85,B 0,C 180,E1 -1888.612,E2 -1888.612} C_VEL
LIN {X 0,Y 580.034,Z 557.5,A -85,B 0,C 180,E1 -1890,E2 -1890} C_VEL
LIN {X 0,Y 580.044,Z 556.911,A -85,B 0,C 180,E1 -1891.389,E2 -1891.389} C_VEL
LIN {X 0,Y 580.04,Z 555.186,A -85,B 0,C 180,E1 -1892.778,E2 -1892.778} C_VEL
LIN {X 0,Y 580.086,Z 552.288,A -85,B 0,C 180,E1 -1894.169,E2 -1894.169} C_VEL
LIN {X 0,Y 580.128,Z 548.162,A -85,B 0,C 180,E1 -1895.562,E2 -1895.562} C_VEL
LIN {X 0,Y 580.138,Z 542.702,A -85,B 0,C 180,E1 -1896.958,E2 -1896.958} C_VEL
LIN {X 0,Y 580.191,Z 535.748,A -85,B 0,C 180,E1 -1898.358,E2 -1898.358} C_VEL
LIN {X 0,Y 580.235,Z 527.088,A -85,B 0,C 180,E1 -1899.763,E2 -1899.763} C_VEL
LIN {X 0,Y 580.343,Z 518.443,A -85,B 0,C 180,E1 -1900.928,E2 -1900.928} C_VEL
LIN {X 0,Y 580.427,Z 508.507,A -85,B 0,C 180,E1 -1902.056,E2 -1902.056} C_VEL
LIN {X 0,Y 580.594,Z 497.384,A -85,B 0,C 180,E1 -1903.119,E2 -1903.119} C_VEL
LIN {X 0,Y 580.776,Z 484.991,A -85,B 0,C 180,E1 -1904.111,E2 -1904.111} C_VEL
LIN {X 0,Y 580.914,Z 471.777,A -85,B 0,C 180,E1 -1904.987,E2 -1904.987} C_VEL
LIN {X 0,Y 581.082,Z 458.599,A -85,B 0,C 180,E1 -1905.701,E2 -1905.701} C_VEL
LIN {X 0,Y 581.234,Z 444.175,A -85,B 0,C 180,E1 -1906.328,E2 -1906.328} C_VEL
LIN {X 0,Y 581.393,Z 429.245,A -85,B 0,C 180,E1 -1906.82,E2 -1906.82} C_VEL
LIN {X 0,Y 581.462,Z 414.084,A -85,B 0,C 180,E1 -1907.173,E2 -1907.173} C_VEL
LIN {X 0,Y 581.502,Z 401.421,A -85,B 0,C 180,E1 -1907.364,E2 -1907.364} C_VEL
LIN {X 0,Y 580.595,Z 396.687,A -85,B 0,C 180,E1 -1907.47,E2 -1907.47} C_VEL
LIN {X 0,Y 580.803,Z 376.47,A -85,B 0,C 180,E1 -1910.358,E2 -1910.358} C_VEL
LIN {X 0,Y 581.01,Z 356.319,A -85,B 0,C 180,E1 -1913.291,E2 -1913.291} C_VEL
LIN {X 0,Y 581.235,Z 338.137,A -85,B 0,C 180,E1 -1915.989,E2 -1915.989} C_VEL
LIN {X 0,Y 581.455,Z 321.45,A -85,B 0,C 180,E1 -1918.518,E2 -1918.518} C_VEL
LIN {X 0,Y 581.63,Z 306.551,A -85,B 0,C 180,E1 -1920.799,E2 -1920.799} C_VEL
LIN {X 0,Y 582.088,Z 291.868,A -85,B 0,C 180,E1 -1923.267,E2 -1923.267} C_VEL
LIN {X 0,Y 582.362,Z 287.055,A -85,B 0,C 180,E1 -1924.137,E2 -1924.137} C_VEL
LIN {X 0,Y 580.487,Z 279.878,A -85,B 0,C 180,E1 -1925.789,E2 -1925.789} C_VEL
LIN {X 0,Y 580.255,Z 278.835,A -85,B 0,C 180,E1 -1926.095,E2 -1926.095} C_VEL
LIN {X 0,Y 580.286,Z 278.83,A -85,B 0,C 180,E1 -1928.147,E2 -1928.147} C_VEL
LIN {X 0,Y 580.297,Z 278.828,A -85,B 0,C 180,E1 -1930.844,E2 -1930.844} C_VEL
LIN {X 0,Y 580.284,Z 278.83,A -85,B 0,C 180,E1 -1933.658,E2 -1933.658} C_VEL
LIN {X 0,Y 580.277,Z 278.833,A -85,B 0,C 180,E1 -1936.61,E2 -1936.61} C_VEL
LIN {X 0,Y 580.295,Z 278.83,A -85,B 0,C 180,E1 -1939.156,E2 -1939.156} C_VEL
LIN {X 0,Y 580.292,Z 278.831,A -85,B 0,C 180,E1 -1941.927,E2 -1941.927} C_VEL
LIN {X 0,Y 580.224,Z 278.865,A -85,B 0,C 180,E1 -1944.451,E2 -1944.451} C_VEL
LIN {X 0,Y 580.293,Z 281.992,A -85,B 0,C 180,E1 -1946.975,E2 -1946.975} C_VEL
LIN {X 0,Y 580.281,Z 284.609,A -85,B 0,C 180,E1 -1949.424,E2 -1949.424} C_VEL
LIN {X 0,Y 580.278,Z 286.914,A -85,B 0,C 180,E1 -1951.813,E2 -1951.813} C_VEL
LIN {X 0,Y 580.208,Z 288.984,A -85,B 0,C 180,E1 -1954.147,E2 -1954.147} C_VEL
LIN {X 0,Y 580.097,Z 291.343,A -85,B 0,C 180,E1 -1957.038,E2 -1957.038} C_VEL
LIN {X 0,Y 580.085,Z 293.997,A -85,B 0,C 180,E1 -1959.43,E2 -1959.43} C_VEL
LIN {X 0,Y 580.039,Z 297.602,A -85,B 0,C 180,E1 -1962.368,E2 -1962.368} C_VEL
LIN {X 0,Y 580.055,Z 300.305,A -85,B 0,C 180,E1 -1964.541,E2 -1964.541} C_VEL
LIN {X 0,Y 580.059,Z 303.008,A -85,B 0,C 180,E1 -1966.691,E2 -1966.691} C_VEL
LIN {X 0,Y 580.056,Z 304.562,A -85,B 0,C 180,E1 -1967.759,E2 -1967.759} C_VEL
LIN {X 0,Y 580.762,Z 309.916,A -85,B 0,C 180,E1 -1967.885,E2 -1967.885} C_VEL
LIN {X 0,Y 580.686,Z 322.96,A -85,B 0,C 180,E1 -1968.26,E2 -1968.26} C_VEL
LIN {X 0,Y 580.595,Z 335.15,A -85,B 0,C 180,E1 -1968.753,E2 -1968.753} C_VEL
LIN {X 0,Y 580.524,Z 346.528,A -85,B 0,C 180,E1 -1969.361,E2 -1969.361} C_VEL
LIN {X 0,Y 580.391,Z 358.167,A -85,B 0,C 180,E1 -1970.152,E2 -1970.152} C_VEL
LIN {X 0,Y 580.308,Z 367.544,A -85,B 0,C 180,E1 -1970.942,E2 -1970.942} C_VEL
LIN {X 0,Y 580.251,Z 376.106,A -85,B 0,C 180,E1 -1971.818,E2 -1971.818} C_VEL
LIN {X 0,Y 580.205,Z 384.419,A -85,B 0,C 180,E1 -1972.868,E2 -1972.868} C_VEL
LIN {X 0,Y 580.14,Z 391.116,A -85,B 0,C 180,E1 -1973.915,E2 -1973.915} C_VEL
LIN {X 0,Y 580.053,Z 397.261,A -85,B 0,C 180,E1 -1975.135,E2 -1975.135} C_VEL
LIN {X 0,Y 580.11,Z 401.25,A -85,B 0,C 180,E1 -1976.18,E2 -1976.18} C_VEL
LIN {X 0,Y 580.043,Z 404.198,A -85,B 0,C 180,E1 -1977.222,E2 -1977.222} C_VEL
LIN {X 0,Y 580.038,Z 405.627,A -85,B 0,C 180,E1 -1977.917,E2 -1977.917} C_VEL
LIN {X 0,Y 580.041,Z 407.255,A -85,B 0,C 180,E1 -1979.306,E2 -1979.306} C_VEL
LIN {X 0,Y 580.038,Z 407.496,A -85,B 0,C 180,E1 -1980,E2 -1980} C_VEL
LIN {X 0,Y 580.04,Z 407.315,A -85,B 0,C 180,E1 -1980.694,E2 -1980.694} C_VEL
LIN {X 0,Y 580.037,Z 405.773,A -85,B 0,C 180,E1 -1982.083,E2 -1982.083} C_VEL
LIN {X 0,Y 580.044,Z 404.413,A -85,B 0,C 180,E1 -1982.778,E2 -1982.778} C_VEL
LIN {X 0,Y 580.11,Z 401.534,A -85,B 0,C 180,E1 -1983.821,E2 -1983.821} C_VEL
LIN {X 0,Y 580.053,Z 397.633,A -85,B 0,C 180,E1 -1984.865,E2 -1984.865} C_VEL
LIN {X 0,Y 580.162,Z 392.603,A -85,B 0,C 180,E1 -1985.91,E2 -1985.91} C_VEL
LIN {X 0,Y 580.158,Z 386.279,A -85,B 0,C 180,E1 -1986.958,E2 -1986.958} C_VEL
LIN {X 0,Y 580.241,Z 378.359,A -85,B 0,C 180,E1 -1988.007,E2 -1988.007} C_VEL
LIN {X 0,Y 580.308,Z 368.51,A -85,B 0,C 180,E1 -1989.058,E2 -1989.058} C_VEL
LIN {X 0,Y 580.413,Z 358.187,A -85,B 0,C 180,E1 -1989.936,E2 -1989.936} C_VEL
LIN {X 0,Y 580.529,Z 346.555,A -85,B 0,C 180,E1 -1990.727,E2 -1990.727} C_VEL
LIN {X 0,Y 580.63,Z 334.801,A -85,B 0,C 180,E1 -1991.352,E2 -1991.352} C_VEL
LIN {X 0,Y 580.684,Z 323.119,A -85,B 0,C 180,E1 -1991.825,E2 -1991.825} C_VEL
LIN {X 0,Y 580.771,Z 309.959,A -85,B 0,C 180,E1 -1992.204,E2 -1992.204} C_VEL
LIN {X 0,Y 580.08,Z 304.333,A -85,B 0,C 180,E1 -1992.352,E2 -1992.352} C_VEL
LIN {X 0,Y 580.045,Z 301.319,A -85,B 0,C 180,E1 -1994.741,E2 -1994.741} C_VEL
LIN {X 0,Y 580.04,Z 298.614,A -85,B 0,C 180,E1 -1996.906,E2 -1996.906} C_VEL
LIN {X 0,Y 580.03,Z 297.975,A -85,B 0,C 180,E1 -1997.421,E2 -1997.421} C_VEL
LIN {X 0,Y 579.376,Z 297.288,A -85,B 0,C 180,E1 -1997.997,E2 -1997.997} C_VEL
LIN {X 0,Y 576.512,Z 296.256,A -85,B 0,C 180,E1 -1998.933,E2 -1998.933} C_VEL
LIN {X 0,Y 574.086,Z 295.443,A -85,B 0,C 180,E1 -1999.686,E2 -1999.686} C_VEL
LIN {X 0,Y 573.05,Z 294.789,A -85,B 0,C 180,E1 -2000.267,E2 -2000.267} C_VEL
LIN {X 0,Y 572.968,Z 294.558,A -85,B 0,C 180,E1 -2000.463,E2 -2000.463} C_VEL
LIN {X 0,Y 572.991,Z 291.694,A -85,B 0,C 180,E1 -2003.11,E2 -2003.11} C_VEL
LIN {X 0,Y 573.038,Z 289.307,A -85,B 0,C 180,E1 -2005.42,E2 -2005.42} C_VEL
LIN {X 0,Y 573.084,Z 286.565,A -85,B 0,C 180,E1 -2007.997,E2 -2007.997} C_VEL
LIN {X 0,Y 573.072,Z 284.168,A -85,B 0,C 180,E1 -2010.186,E2 -2010.186} C_VEL
LIN {X 0,Y 573.034,Z 281.39,A -85,B 0,C 180,E1 -2012.659,E2 -2012.659} C_VEL
LIN {X 0,Y 573.081,Z 279.729,A -85,B 0,C 180,E1 -2014.341,E2 -2014.341} C_VEL
LIN {X 0,Y 573.255,Z 279.707,A -85,B 0,C 180,E1 -2017.166,E2 -2017.166} C_VEL
LIN {X 0,Y 573.251,Z 279.7,A -85,B 0,C 180,E1 -2019.607,E2 -2019.607} C_VEL
LIN {X 0,Y 573.242,Z 279.707,A -85,B 0,C 180,E1 -2022.641,E2 -2022.641} C_VEL
LIN {X 0,Y 573.219,Z 279.705,A -85,B 0,C 180,E1 -2025.665,E2 -2025.665} C_VEL
LIN {X 0,Y 573.196,Z 279.71,A -85,B 0,C 180,E1 -2028.411,E2 -2028.411} C_VEL
LIN {X 0,Y 573.201,Z 279.711,A -85,B 0,C 180,E1 -2029.48,E2 -2029.48} C_VEL
LIN {X 0,Y 573.206,Z 282.467,A -85,B 0,C 180,E1 -2031.295,E2 -2031.295} C_VEL
LIN {X 0,Y 573.177,Z 286.626,A -85,B 0,C 180,E1 -2033.945,E2 -2033.945} C_VEL
LIN {X 0,Y 573.149,Z 290.263,A -85,B 0,C 180,E1 -2036.51,E2 -2036.51} C_VEL
